   // GBK_TO_UNICODE[34568] := 16#E38B;
   // GBK_TO_UNICODE[34569] := 16#9292;
   // GBK_TO_UNICODE[34570] := 16#E38C;
   // GBK_TO_UNICODE[34571] := 16#9293;
   // GBK_TO_UNICODE[34572] := 16#E38D;
   // GBK_TO_UNICODE[34573] := 16#9294;
   // GBK_TO_UNICODE[34574] := 16#E38E;
   // GBK_TO_UNICODE[34575] := 16#9295;
   // GBK_TO_UNICODE[34576] := 16#E38F;
   // GBK_TO_UNICODE[34577] := 16#9296;
   // GBK_TO_UNICODE[34578] := 16#E390;
   // GBK_TO_UNICODE[34579] := 16#9297;
   // GBK_TO_UNICODE[34580] := 16#E391;
   // GBK_TO_UNICODE[34581] := 16#9298;
   // GBK_TO_UNICODE[34582] := 16#E392;
   // GBK_TO_UNICODE[34583] := 16#9299;
   // GBK_TO_UNICODE[34584] := 16#E393;
   // GBK_TO_UNICODE[34585] := 16#929A;
   // GBK_TO_UNICODE[34586] := 16#E394;
   // GBK_TO_UNICODE[34587] := 16#929B;
   // GBK_TO_UNICODE[34588] := 16#E395;
   // GBK_TO_UNICODE[34589] := 16#929C;
   // GBK_TO_UNICODE[34590] := 16#E396;
   // GBK_TO_UNICODE[34591] := 16#929D;
   // GBK_TO_UNICODE[34592] := 16#E397;
   // GBK_TO_UNICODE[34593] := 16#929E;
   // GBK_TO_UNICODE[34594] := 16#E398;
   // GBK_TO_UNICODE[34595] := 16#929F;
   // GBK_TO_UNICODE[34596] := 16#E399;
   // GBK_TO_UNICODE[34597] := 16#92A0;
   // GBK_TO_UNICODE[34598] := 16#E39A;
   // GBK_TO_UNICODE[34599] := 16#92A1;
   // GBK_TO_UNICODE[34600] := 16#E39B;
   // GBK_TO_UNICODE[34601] := 16#92A2;
   // GBK_TO_UNICODE[34602] := 16#E39C;
   // GBK_TO_UNICODE[34603] := 16#92A3;
   // GBK_TO_UNICODE[34604] := 16#E39D;
   // GBK_TO_UNICODE[34605] := 16#92A4;
   // GBK_TO_UNICODE[34606] := 16#E39E;
   // GBK_TO_UNICODE[34607] := 16#92A5;
   // GBK_TO_UNICODE[34608] := 16#E39F;
   // GBK_TO_UNICODE[34609] := 16#92A6;
   // GBK_TO_UNICODE[34610] := 16#E3A0;
   // GBK_TO_UNICODE[34611] := 16#92A7;
   // GBK_TO_UNICODE[34612] := 16#E3A1;
   // GBK_TO_UNICODE[34613] := 16#606A;
   // GBK_TO_UNICODE[34614] := 16#E3A2;
   // GBK_TO_UNICODE[34615] := 16#607D;
   // GBK_TO_UNICODE[34616] := 16#E3A3;
   // GBK_TO_UNICODE[34617] := 16#6096;
   // GBK_TO_UNICODE[34618] := 16#E3A4;
   // GBK_TO_UNICODE[34619] := 16#609A;
   // GBK_TO_UNICODE[34620] := 16#E3A5;
   // GBK_TO_UNICODE[34621] := 16#60AD;
   // GBK_TO_UNICODE[34622] := 16#E3A6;
   // GBK_TO_UNICODE[34623] := 16#609D;
   // GBK_TO_UNICODE[34624] := 16#E3A7;
   // GBK_TO_UNICODE[34625] := 16#6083;
   // GBK_TO_UNICODE[34626] := 16#E3A8;
   // GBK_TO_UNICODE[34627] := 16#6092;
   // GBK_TO_UNICODE[34628] := 16#E3A9;
   // GBK_TO_UNICODE[34629] := 16#608C;
   // GBK_TO_UNICODE[34630] := 16#E3AA;
   // GBK_TO_UNICODE[34631] := 16#609B;
   // GBK_TO_UNICODE[34632] := 16#E3AB;
   // GBK_TO_UNICODE[34633] := 16#60EC;
   // GBK_TO_UNICODE[34634] := 16#E3AC;
   // GBK_TO_UNICODE[34635] := 16#60BB;
   // GBK_TO_UNICODE[34636] := 16#E3AD;
   // GBK_TO_UNICODE[34637] := 16#60B1;
   // GBK_TO_UNICODE[34638] := 16#E3AE;
   // GBK_TO_UNICODE[34639] := 16#60DD;
   // GBK_TO_UNICODE[34640] := 16#E3AF;
   // GBK_TO_UNICODE[34641] := 16#60D8;
   // GBK_TO_UNICODE[34642] := 16#E3B0;
   // GBK_TO_UNICODE[34643] := 16#60C6;
   // GBK_TO_UNICODE[34644] := 16#E3B1;
   // GBK_TO_UNICODE[34645] := 16#60DA;
   // GBK_TO_UNICODE[34646] := 16#E3B2;
   // GBK_TO_UNICODE[34647] := 16#60B4;
   // GBK_TO_UNICODE[34648] := 16#E3B3;
   // GBK_TO_UNICODE[34649] := 16#6120;
   // GBK_TO_UNICODE[34650] := 16#E3B4;
   // GBK_TO_UNICODE[34651] := 16#6126;
   // GBK_TO_UNICODE[34652] := 16#E3B5;
   // GBK_TO_UNICODE[34653] := 16#6115;
   // GBK_TO_UNICODE[34654] := 16#E3B6;
   // GBK_TO_UNICODE[34655] := 16#6123;
   // GBK_TO_UNICODE[34656] := 16#E3B7;
   // GBK_TO_UNICODE[34657] := 16#60F4;
   // GBK_TO_UNICODE[34658] := 16#E3B8;
   // GBK_TO_UNICODE[34659] := 16#6100;
   // GBK_TO_UNICODE[34660] := 16#E3B9;
   // GBK_TO_UNICODE[34661] := 16#610E;
   // GBK_TO_UNICODE[34662] := 16#E3BA;
   // GBK_TO_UNICODE[34663] := 16#612B;
   // GBK_TO_UNICODE[34664] := 16#E3BB;
   // GBK_TO_UNICODE[34665] := 16#614A;
   // GBK_TO_UNICODE[34666] := 16#E3BC;
   // GBK_TO_UNICODE[34667] := 16#6175;
   // GBK_TO_UNICODE[34668] := 16#E3BD;
   // GBK_TO_UNICODE[34669] := 16#61AC;
   // GBK_TO_UNICODE[34670] := 16#E3BE;
   // GBK_TO_UNICODE[34671] := 16#6194;
   // GBK_TO_UNICODE[34672] := 16#E3BF;
   // GBK_TO_UNICODE[34673] := 16#61A7;
   // GBK_TO_UNICODE[34674] := 16#E3C0;
   // GBK_TO_UNICODE[34675] := 16#61B7;
   // GBK_TO_UNICODE[34676] := 16#E3C1;
   // GBK_TO_UNICODE[34677] := 16#61D4;
   // GBK_TO_UNICODE[34678] := 16#E3C2;
   // GBK_TO_UNICODE[34679] := 16#61F5;
   // GBK_TO_UNICODE[34680] := 16#E3C3;
   // GBK_TO_UNICODE[34681] := 16#5FDD;
   // GBK_TO_UNICODE[34682] := 16#E3C4;
   // GBK_TO_UNICODE[34683] := 16#96B3;
   // GBK_TO_UNICODE[34684] := 16#E3C5;
   // GBK_TO_UNICODE[34685] := 16#95E9;
   // GBK_TO_UNICODE[34686] := 16#E3C6;
   // GBK_TO_UNICODE[34687] := 16#95EB;
   // GBK_TO_UNICODE[34688] := 16#E3C7;
   // GBK_TO_UNICODE[34689] := 16#95F1;
   // GBK_TO_UNICODE[34690] := 16#E3C8;
   // GBK_TO_UNICODE[34691] := 16#95F3;
   // GBK_TO_UNICODE[34692] := 16#E3C9;
   // GBK_TO_UNICODE[34693] := 16#95F5;
   // GBK_TO_UNICODE[34694] := 16#E3CA;
   // GBK_TO_UNICODE[34695] := 16#95F6;
   // GBK_TO_UNICODE[34696] := 16#E3CB;
   // GBK_TO_UNICODE[34697] := 16#95FC;
   // GBK_TO_UNICODE[34698] := 16#E3CC;
   // GBK_TO_UNICODE[34699] := 16#95FE;
   // GBK_TO_UNICODE[34700] := 16#E3CD;
   // GBK_TO_UNICODE[34701] := 16#9603;
   // GBK_TO_UNICODE[34702] := 16#E3CE;
   // GBK_TO_UNICODE[34703] := 16#9604;
   // GBK_TO_UNICODE[34704] := 16#E3CF;
   // GBK_TO_UNICODE[34705] := 16#9606;
   // GBK_TO_UNICODE[34706] := 16#E3D0;
   // GBK_TO_UNICODE[34707] := 16#9608;
   // GBK_TO_UNICODE[34708] := 16#E3D1;
   // GBK_TO_UNICODE[34709] := 16#960A;
   // GBK_TO_UNICODE[34710] := 16#E3D2;
   // GBK_TO_UNICODE[34711] := 16#960B;
   // GBK_TO_UNICODE[34712] := 16#E3D3;
   // GBK_TO_UNICODE[34713] := 16#960C;
   // GBK_TO_UNICODE[34714] := 16#E3D4;
   // GBK_TO_UNICODE[34715] := 16#960D;
   // GBK_TO_UNICODE[34716] := 16#E3D5;
   // GBK_TO_UNICODE[34717] := 16#960F;
   // GBK_TO_UNICODE[34718] := 16#E3D6;
   // GBK_TO_UNICODE[34719] := 16#9612;
   // GBK_TO_UNICODE[34720] := 16#E3D7;
   // GBK_TO_UNICODE[34721] := 16#9615;
   // GBK_TO_UNICODE[34722] := 16#E3D8;
   // GBK_TO_UNICODE[34723] := 16#9616;
   // GBK_TO_UNICODE[34724] := 16#E3D9;
   // GBK_TO_UNICODE[34725] := 16#9617;
   // GBK_TO_UNICODE[34726] := 16#E3DA;
   // GBK_TO_UNICODE[34727] := 16#9619;
   // GBK_TO_UNICODE[34728] := 16#E3DB;
   // GBK_TO_UNICODE[34729] := 16#961A;
   // GBK_TO_UNICODE[34730] := 16#E3DC;
   // GBK_TO_UNICODE[34731] := 16#4E2C;
   // GBK_TO_UNICODE[34732] := 16#E3DD;
   // GBK_TO_UNICODE[34733] := 16#723F;
   // GBK_TO_UNICODE[34734] := 16#E3DE;
   // GBK_TO_UNICODE[34735] := 16#6215;
   // GBK_TO_UNICODE[34736] := 16#E3DF;
   // GBK_TO_UNICODE[34737] := 16#6C35;
   // GBK_TO_UNICODE[34738] := 16#E3E0;
   // GBK_TO_UNICODE[34739] := 16#6C54;
   // GBK_TO_UNICODE[34740] := 16#E3E1;
   // GBK_TO_UNICODE[34741] := 16#6C5C;
   // GBK_TO_UNICODE[34742] := 16#E3E2;
   // GBK_TO_UNICODE[34743] := 16#6C4A;
   // GBK_TO_UNICODE[34744] := 16#E3E3;
   // GBK_TO_UNICODE[34745] := 16#6CA3;
   // GBK_TO_UNICODE[34746] := 16#E3E4;
   // GBK_TO_UNICODE[34747] := 16#6C85;
   // GBK_TO_UNICODE[34748] := 16#E3E5;
   // GBK_TO_UNICODE[34749] := 16#6C90;
   // GBK_TO_UNICODE[34750] := 16#E3E6;
   // GBK_TO_UNICODE[34751] := 16#6C94;
   // GBK_TO_UNICODE[34752] := 16#E3E7;
   // GBK_TO_UNICODE[34753] := 16#6C8C;
   // GBK_TO_UNICODE[34754] := 16#E3E8;
   // GBK_TO_UNICODE[34755] := 16#6C68;
   // GBK_TO_UNICODE[34756] := 16#E3E9;
   // GBK_TO_UNICODE[34757] := 16#6C69;
   // GBK_TO_UNICODE[34758] := 16#E3EA;
   // GBK_TO_UNICODE[34759] := 16#6C74;
   // GBK_TO_UNICODE[34760] := 16#E3EB;
   // GBK_TO_UNICODE[34761] := 16#6C76;
   // GBK_TO_UNICODE[34762] := 16#E3EC;
   // GBK_TO_UNICODE[34763] := 16#6C86;
   // GBK_TO_UNICODE[34764] := 16#E3ED;
   // GBK_TO_UNICODE[34765] := 16#6CA9;
   // GBK_TO_UNICODE[34766] := 16#E3EE;
   // GBK_TO_UNICODE[34767] := 16#6CD0;
   // GBK_TO_UNICODE[34768] := 16#E3EF;
   // GBK_TO_UNICODE[34769] := 16#6CD4;
   // GBK_TO_UNICODE[34770] := 16#E3F0;
   // GBK_TO_UNICODE[34771] := 16#6CAD;
   // GBK_TO_UNICODE[34772] := 16#E3F1;
   // GBK_TO_UNICODE[34773] := 16#6CF7;
   // GBK_TO_UNICODE[34774] := 16#E3F2;
   // GBK_TO_UNICODE[34775] := 16#6CF8;
   // GBK_TO_UNICODE[34776] := 16#E3F3;
   // GBK_TO_UNICODE[34777] := 16#6CF1;
   // GBK_TO_UNICODE[34778] := 16#E3F4;
   // GBK_TO_UNICODE[34779] := 16#6CD7;
   // GBK_TO_UNICODE[34780] := 16#E3F5;
   // GBK_TO_UNICODE[34781] := 16#6CB2;
   // GBK_TO_UNICODE[34782] := 16#E3F6;
   // GBK_TO_UNICODE[34783] := 16#6CE0;
   // GBK_TO_UNICODE[34784] := 16#E3F7;
   // GBK_TO_UNICODE[34785] := 16#6CD6;
   // GBK_TO_UNICODE[34786] := 16#E3F8;
   // GBK_TO_UNICODE[34787] := 16#6CFA;
   // GBK_TO_UNICODE[34788] := 16#E3F9;
   // GBK_TO_UNICODE[34789] := 16#6CEB;
   // GBK_TO_UNICODE[34790] := 16#E3FA;
   // GBK_TO_UNICODE[34791] := 16#6CEE;
   // GBK_TO_UNICODE[34792] := 16#E3FB;
   // GBK_TO_UNICODE[34793] := 16#6CB1;
   // GBK_TO_UNICODE[34794] := 16#E3FC;
   // GBK_TO_UNICODE[34795] := 16#6CD3;
   // GBK_TO_UNICODE[34796] := 16#E3FD;
   // GBK_TO_UNICODE[34797] := 16#6CEF;
   // GBK_TO_UNICODE[34798] := 16#E3FE;
   // GBK_TO_UNICODE[34799] := 16#6CFE;
   // GBK_TO_UNICODE[34800] := 16#E440;
   // GBK_TO_UNICODE[34801] := 16#92A8;
   // GBK_TO_UNICODE[34802] := 16#E441;
   // GBK_TO_UNICODE[34803] := 16#92A9;
   // GBK_TO_UNICODE[34804] := 16#E442;
   // GBK_TO_UNICODE[34805] := 16#92AA;
   // GBK_TO_UNICODE[34806] := 16#E443;
   // GBK_TO_UNICODE[34807] := 16#92AB;
   // GBK_TO_UNICODE[34808] := 16#E444;
   // GBK_TO_UNICODE[34809] := 16#92AC;
   // GBK_TO_UNICODE[34810] := 16#E445;
   // GBK_TO_UNICODE[34811] := 16#92AD;
   // GBK_TO_UNICODE[34812] := 16#E446;
   // GBK_TO_UNICODE[34813] := 16#92AF;
   // GBK_TO_UNICODE[34814] := 16#E447;
   // GBK_TO_UNICODE[34815] := 16#92B0;
   // GBK_TO_UNICODE[34816] := 16#E448;
   // GBK_TO_UNICODE[34817] := 16#92B1;
   // GBK_TO_UNICODE[34818] := 16#E449;
   // GBK_TO_UNICODE[34819] := 16#92B2;
   // GBK_TO_UNICODE[34820] := 16#E44A;
   // GBK_TO_UNICODE[34821] := 16#92B3;
   // GBK_TO_UNICODE[34822] := 16#E44B;
   // GBK_TO_UNICODE[34823] := 16#92B4;
   // GBK_TO_UNICODE[34824] := 16#E44C;
   // GBK_TO_UNICODE[34825] := 16#92B5;
   // GBK_TO_UNICODE[34826] := 16#E44D;
   // GBK_TO_UNICODE[34827] := 16#92B6;
   // GBK_TO_UNICODE[34828] := 16#E44E;
   // GBK_TO_UNICODE[34829] := 16#92B7;
   // GBK_TO_UNICODE[34830] := 16#E44F;
   // GBK_TO_UNICODE[34831] := 16#92B8;
   // GBK_TO_UNICODE[34832] := 16#E450;
   // GBK_TO_UNICODE[34833] := 16#92B9;
   // GBK_TO_UNICODE[34834] := 16#E451;
   // GBK_TO_UNICODE[34835] := 16#92BA;
   // GBK_TO_UNICODE[34836] := 16#E452;
   // GBK_TO_UNICODE[34837] := 16#92BB;
   // GBK_TO_UNICODE[34838] := 16#E453;
   // GBK_TO_UNICODE[34839] := 16#92BC;
   // GBK_TO_UNICODE[34840] := 16#E454;
   // GBK_TO_UNICODE[34841] := 16#92BD;
   // GBK_TO_UNICODE[34842] := 16#E455;
   // GBK_TO_UNICODE[34843] := 16#92BE;
   // GBK_TO_UNICODE[34844] := 16#E456;
   // GBK_TO_UNICODE[34845] := 16#92BF;
   // GBK_TO_UNICODE[34846] := 16#E457;
   // GBK_TO_UNICODE[34847] := 16#92C0;
   // GBK_TO_UNICODE[34848] := 16#E458;
   // GBK_TO_UNICODE[34849] := 16#92C1;
   // GBK_TO_UNICODE[34850] := 16#E459;
   // GBK_TO_UNICODE[34851] := 16#92C2;
   // GBK_TO_UNICODE[34852] := 16#E45A;
   // GBK_TO_UNICODE[34853] := 16#92C3;
   // GBK_TO_UNICODE[34854] := 16#E45B;
   // GBK_TO_UNICODE[34855] := 16#92C4;
   // GBK_TO_UNICODE[34856] := 16#E45C;
   // GBK_TO_UNICODE[34857] := 16#92C5;
   // GBK_TO_UNICODE[34858] := 16#E45D;
   // GBK_TO_UNICODE[34859] := 16#92C6;
   // GBK_TO_UNICODE[34860] := 16#E45E;
   // GBK_TO_UNICODE[34861] := 16#92C7;
   // GBK_TO_UNICODE[34862] := 16#E45F;
   // GBK_TO_UNICODE[34863] := 16#92C9;
   // GBK_TO_UNICODE[34864] := 16#E460;
   // GBK_TO_UNICODE[34865] := 16#92CA;
   // GBK_TO_UNICODE[34866] := 16#E461;
   // GBK_TO_UNICODE[34867] := 16#92CB;
   // GBK_TO_UNICODE[34868] := 16#E462;
   // GBK_TO_UNICODE[34869] := 16#92CC;
   // GBK_TO_UNICODE[34870] := 16#E463;
   // GBK_TO_UNICODE[34871] := 16#92CD;
   // GBK_TO_UNICODE[34872] := 16#E464;
   // GBK_TO_UNICODE[34873] := 16#92CE;
   // GBK_TO_UNICODE[34874] := 16#E465;
   // GBK_TO_UNICODE[34875] := 16#92CF;
   // GBK_TO_UNICODE[34876] := 16#E466;
   // GBK_TO_UNICODE[34877] := 16#92D0;
   // GBK_TO_UNICODE[34878] := 16#E467;
   // GBK_TO_UNICODE[34879] := 16#92D1;
   // GBK_TO_UNICODE[34880] := 16#E468;
   // GBK_TO_UNICODE[34881] := 16#92D2;
   // GBK_TO_UNICODE[34882] := 16#E469;
   // GBK_TO_UNICODE[34883] := 16#92D3;
   // GBK_TO_UNICODE[34884] := 16#E46A;
   // GBK_TO_UNICODE[34885] := 16#92D4;
   // GBK_TO_UNICODE[34886] := 16#E46B;
   // GBK_TO_UNICODE[34887] := 16#92D5;
   // GBK_TO_UNICODE[34888] := 16#E46C;
   // GBK_TO_UNICODE[34889] := 16#92D6;
   // GBK_TO_UNICODE[34890] := 16#E46D;
   // GBK_TO_UNICODE[34891] := 16#92D7;
   // GBK_TO_UNICODE[34892] := 16#E46E;
   // GBK_TO_UNICODE[34893] := 16#92D8;
   // GBK_TO_UNICODE[34894] := 16#E46F;
   // GBK_TO_UNICODE[34895] := 16#92D9;
   // GBK_TO_UNICODE[34896] := 16#E470;
   // GBK_TO_UNICODE[34897] := 16#92DA;
   // GBK_TO_UNICODE[34898] := 16#E471;
   // GBK_TO_UNICODE[34899] := 16#92DB;
   // GBK_TO_UNICODE[34900] := 16#E472;
   // GBK_TO_UNICODE[34901] := 16#92DC;
   // GBK_TO_UNICODE[34902] := 16#E473;
   // GBK_TO_UNICODE[34903] := 16#92DD;
   // GBK_TO_UNICODE[34904] := 16#E474;
   // GBK_TO_UNICODE[34905] := 16#92DE;
   // GBK_TO_UNICODE[34906] := 16#E475;
   // GBK_TO_UNICODE[34907] := 16#92DF;
   // GBK_TO_UNICODE[34908] := 16#E476;
   // GBK_TO_UNICODE[34909] := 16#92E0;
   // GBK_TO_UNICODE[34910] := 16#E477;
   // GBK_TO_UNICODE[34911] := 16#92E1;
   // GBK_TO_UNICODE[34912] := 16#E478;
   // GBK_TO_UNICODE[34913] := 16#92E2;
   // GBK_TO_UNICODE[34914] := 16#E479;
   // GBK_TO_UNICODE[34915] := 16#92E3;
   // GBK_TO_UNICODE[34916] := 16#E47A;
   // GBK_TO_UNICODE[34917] := 16#92E4;
   // GBK_TO_UNICODE[34918] := 16#E47B;
   // GBK_TO_UNICODE[34919] := 16#92E5;
   // GBK_TO_UNICODE[34920] := 16#E47C;
   // GBK_TO_UNICODE[34921] := 16#92E6;
   // GBK_TO_UNICODE[34922] := 16#E47D;
   // GBK_TO_UNICODE[34923] := 16#92E7;
   // GBK_TO_UNICODE[34924] := 16#E47E;
   // GBK_TO_UNICODE[34925] := 16#92E8;
   // GBK_TO_UNICODE[34926] := 16#E480;
   // GBK_TO_UNICODE[34927] := 16#92E9;
   // GBK_TO_UNICODE[34928] := 16#E481;
   // GBK_TO_UNICODE[34929] := 16#92EA;
   // GBK_TO_UNICODE[34930] := 16#E482;
   // GBK_TO_UNICODE[34931] := 16#92EB;
   // GBK_TO_UNICODE[34932] := 16#E483;
   // GBK_TO_UNICODE[34933] := 16#92EC;
   // GBK_TO_UNICODE[34934] := 16#E484;
   // GBK_TO_UNICODE[34935] := 16#92ED;
   // GBK_TO_UNICODE[34936] := 16#E485;
   // GBK_TO_UNICODE[34937] := 16#92EE;
   // GBK_TO_UNICODE[34938] := 16#E486;
   // GBK_TO_UNICODE[34939] := 16#92EF;
   // GBK_TO_UNICODE[34940] := 16#E487;
   // GBK_TO_UNICODE[34941] := 16#92F0;
   // GBK_TO_UNICODE[34942] := 16#E488;
   // GBK_TO_UNICODE[34943] := 16#92F1;
   // GBK_TO_UNICODE[34944] := 16#E489;
   // GBK_TO_UNICODE[34945] := 16#92F2;
   // GBK_TO_UNICODE[34946] := 16#E48A;
   // GBK_TO_UNICODE[34947] := 16#92F3;
   // GBK_TO_UNICODE[34948] := 16#E48B;
   // GBK_TO_UNICODE[34949] := 16#92F4;
   // GBK_TO_UNICODE[34950] := 16#E48C;
   // GBK_TO_UNICODE[34951] := 16#92F5;
   // GBK_TO_UNICODE[34952] := 16#E48D;
   // GBK_TO_UNICODE[34953] := 16#92F6;
   // GBK_TO_UNICODE[34954] := 16#E48E;
   // GBK_TO_UNICODE[34955] := 16#92F7;
   // GBK_TO_UNICODE[34956] := 16#E48F;
   // GBK_TO_UNICODE[34957] := 16#92F8;
   // GBK_TO_UNICODE[34958] := 16#E490;
   // GBK_TO_UNICODE[34959] := 16#92F9;
   // GBK_TO_UNICODE[34960] := 16#E491;
   // GBK_TO_UNICODE[34961] := 16#92FA;
   // GBK_TO_UNICODE[34962] := 16#E492;
   // GBK_TO_UNICODE[34963] := 16#92FB;
   // GBK_TO_UNICODE[34964] := 16#E493;
   // GBK_TO_UNICODE[34965] := 16#92FC;
   // GBK_TO_UNICODE[34966] := 16#E494;
   // GBK_TO_UNICODE[34967] := 16#92FD;
   // GBK_TO_UNICODE[34968] := 16#E495;
   // GBK_TO_UNICODE[34969] := 16#92FE;
   // GBK_TO_UNICODE[34970] := 16#E496;
   // GBK_TO_UNICODE[34971] := 16#92FF;
   // GBK_TO_UNICODE[34972] := 16#E497;
   // GBK_TO_UNICODE[34973] := 16#9300;
   // GBK_TO_UNICODE[34974] := 16#E498;
   // GBK_TO_UNICODE[34975] := 16#9301;
   // GBK_TO_UNICODE[34976] := 16#E499;
   // GBK_TO_UNICODE[34977] := 16#9302;
   // GBK_TO_UNICODE[34978] := 16#E49A;
   // GBK_TO_UNICODE[34979] := 16#9303;
   // GBK_TO_UNICODE[34980] := 16#E49B;
   // GBK_TO_UNICODE[34981] := 16#9304;
   // GBK_TO_UNICODE[34982] := 16#E49C;
   // GBK_TO_UNICODE[34983] := 16#9305;
   // GBK_TO_UNICODE[34984] := 16#E49D;
   // GBK_TO_UNICODE[34985] := 16#9306;
   // GBK_TO_UNICODE[34986] := 16#E49E;
   // GBK_TO_UNICODE[34987] := 16#9307;
   // GBK_TO_UNICODE[34988] := 16#E49F;
   // GBK_TO_UNICODE[34989] := 16#9308;
   // GBK_TO_UNICODE[34990] := 16#E4A0;
   // GBK_TO_UNICODE[34991] := 16#9309;
   // GBK_TO_UNICODE[34992] := 16#E4A1;
   // GBK_TO_UNICODE[34993] := 16#6D39;
   // GBK_TO_UNICODE[34994] := 16#E4A2;
   // GBK_TO_UNICODE[34995] := 16#6D27;
   // GBK_TO_UNICODE[34996] := 16#E4A3;
   // GBK_TO_UNICODE[34997] := 16#6D0C;
   // GBK_TO_UNICODE[34998] := 16#E4A4;
   // GBK_TO_UNICODE[34999] := 16#6D43;
   // GBK_TO_UNICODE[35000] := 16#E4A5;
   // GBK_TO_UNICODE[35001] := 16#6D48;
   // GBK_TO_UNICODE[35002] := 16#E4A6;
   // GBK_TO_UNICODE[35003] := 16#6D07;
   // GBK_TO_UNICODE[35004] := 16#E4A7;
   // GBK_TO_UNICODE[35005] := 16#6D04;
   // GBK_TO_UNICODE[35006] := 16#E4A8;
   // GBK_TO_UNICODE[35007] := 16#6D19;
   // GBK_TO_UNICODE[35008] := 16#E4A9;
   // GBK_TO_UNICODE[35009] := 16#6D0E;
   // GBK_TO_UNICODE[35010] := 16#E4AA;
   // GBK_TO_UNICODE[35011] := 16#6D2B;
   // GBK_TO_UNICODE[35012] := 16#E4AB;
   // GBK_TO_UNICODE[35013] := 16#6D4D;
   // GBK_TO_UNICODE[35014] := 16#E4AC;
   // GBK_TO_UNICODE[35015] := 16#6D2E;
   // GBK_TO_UNICODE[35016] := 16#E4AD;
   // GBK_TO_UNICODE[35017] := 16#6D35;
   // GBK_TO_UNICODE[35018] := 16#E4AE;
   // GBK_TO_UNICODE[35019] := 16#6D1A;
   // GBK_TO_UNICODE[35020] := 16#E4AF;
   // GBK_TO_UNICODE[35021] := 16#6D4F;
   // GBK_TO_UNICODE[35022] := 16#E4B0;
   // GBK_TO_UNICODE[35023] := 16#6D52;
   // GBK_TO_UNICODE[35024] := 16#E4B1;
   // GBK_TO_UNICODE[35025] := 16#6D54;
   // GBK_TO_UNICODE[35026] := 16#E4B2;
   // GBK_TO_UNICODE[35027] := 16#6D33;
   // GBK_TO_UNICODE[35028] := 16#E4B3;
   // GBK_TO_UNICODE[35029] := 16#6D91;
   // GBK_TO_UNICODE[35030] := 16#E4B4;
   // GBK_TO_UNICODE[35031] := 16#6D6F;
   // GBK_TO_UNICODE[35032] := 16#E4B5;
   // GBK_TO_UNICODE[35033] := 16#6D9E;
   // GBK_TO_UNICODE[35034] := 16#E4B6;
   // GBK_TO_UNICODE[35035] := 16#6DA0;
   // GBK_TO_UNICODE[35036] := 16#E4B7;
   // GBK_TO_UNICODE[35037] := 16#6D5E;
   // GBK_TO_UNICODE[35038] := 16#E4B8;
   // GBK_TO_UNICODE[35039] := 16#6D93;
   // GBK_TO_UNICODE[35040] := 16#E4B9;
   // GBK_TO_UNICODE[35041] := 16#6D94;
   // GBK_TO_UNICODE[35042] := 16#E4BA;
   // GBK_TO_UNICODE[35043] := 16#6D5C;
   // GBK_TO_UNICODE[35044] := 16#E4BB;
   // GBK_TO_UNICODE[35045] := 16#6D60;
   // GBK_TO_UNICODE[35046] := 16#E4BC;
   // GBK_TO_UNICODE[35047] := 16#6D7C;
   // GBK_TO_UNICODE[35048] := 16#E4BD;
   // GBK_TO_UNICODE[35049] := 16#6D63;
   // GBK_TO_UNICODE[35050] := 16#E4BE;
   // GBK_TO_UNICODE[35051] := 16#6E1A;
   // GBK_TO_UNICODE[35052] := 16#E4BF;
   // GBK_TO_UNICODE[35053] := 16#6DC7;
   // GBK_TO_UNICODE[35054] := 16#E4C0;
   // GBK_TO_UNICODE[35055] := 16#6DC5;
   // GBK_TO_UNICODE[35056] := 16#E4C1;
   // GBK_TO_UNICODE[35057] := 16#6DDE;
   // GBK_TO_UNICODE[35058] := 16#E4C2;
   // GBK_TO_UNICODE[35059] := 16#6E0E;
   // GBK_TO_UNICODE[35060] := 16#E4C3;
   // GBK_TO_UNICODE[35061] := 16#6DBF;
   // GBK_TO_UNICODE[35062] := 16#E4C4;
   // GBK_TO_UNICODE[35063] := 16#6DE0;
   // GBK_TO_UNICODE[35064] := 16#E4C5;
   // GBK_TO_UNICODE[35065] := 16#6E11;
   // GBK_TO_UNICODE[35066] := 16#E4C6;
   // GBK_TO_UNICODE[35067] := 16#6DE6;
   // GBK_TO_UNICODE[35068] := 16#E4C7;
   // GBK_TO_UNICODE[35069] := 16#6DDD;
   // GBK_TO_UNICODE[35070] := 16#E4C8;
   // GBK_TO_UNICODE[35071] := 16#6DD9;
   // GBK_TO_UNICODE[35072] := 16#E4C9;
   // GBK_TO_UNICODE[35073] := 16#6E16;
   // GBK_TO_UNICODE[35074] := 16#E4CA;
   // GBK_TO_UNICODE[35075] := 16#6DAB;
   // GBK_TO_UNICODE[35076] := 16#E4CB;
   // GBK_TO_UNICODE[35077] := 16#6E0C;
   // GBK_TO_UNICODE[35078] := 16#E4CC;
   // GBK_TO_UNICODE[35079] := 16#6DAE;
   // GBK_TO_UNICODE[35080] := 16#E4CD;
   // GBK_TO_UNICODE[35081] := 16#6E2B;
   // GBK_TO_UNICODE[35082] := 16#E4CE;
   // GBK_TO_UNICODE[35083] := 16#6E6E;
   // GBK_TO_UNICODE[35084] := 16#E4CF;
   // GBK_TO_UNICODE[35085] := 16#6E4E;
   // GBK_TO_UNICODE[35086] := 16#E4D0;
   // GBK_TO_UNICODE[35087] := 16#6E6B;
   // GBK_TO_UNICODE[35088] := 16#E4D1;
   // GBK_TO_UNICODE[35089] := 16#6EB2;
   // GBK_TO_UNICODE[35090] := 16#E4D2;
   // GBK_TO_UNICODE[35091] := 16#6E5F;
   // GBK_TO_UNICODE[35092] := 16#E4D3;
   // GBK_TO_UNICODE[35093] := 16#6E86;
   // GBK_TO_UNICODE[35094] := 16#E4D4;
   // GBK_TO_UNICODE[35095] := 16#6E53;
   // GBK_TO_UNICODE[35096] := 16#E4D5;
   // GBK_TO_UNICODE[35097] := 16#6E54;
   // GBK_TO_UNICODE[35098] := 16#E4D6;
   // GBK_TO_UNICODE[35099] := 16#6E32;
   // GBK_TO_UNICODE[35100] := 16#E4D7;
   // GBK_TO_UNICODE[35101] := 16#6E25;
   // GBK_TO_UNICODE[35102] := 16#E4D8;
   // GBK_TO_UNICODE[35103] := 16#6E44;
   // GBK_TO_UNICODE[35104] := 16#E4D9;
   // GBK_TO_UNICODE[35105] := 16#6EDF;
   // GBK_TO_UNICODE[35106] := 16#E4DA;
   // GBK_TO_UNICODE[35107] := 16#6EB1;
   // GBK_TO_UNICODE[35108] := 16#E4DB;
   // GBK_TO_UNICODE[35109] := 16#6E98;
   // GBK_TO_UNICODE[35110] := 16#E4DC;
   // GBK_TO_UNICODE[35111] := 16#6EE0;
   // GBK_TO_UNICODE[35112] := 16#E4DD;
   // GBK_TO_UNICODE[35113] := 16#6F2D;
   // GBK_TO_UNICODE[35114] := 16#E4DE;
   // GBK_TO_UNICODE[35115] := 16#6EE2;
   // GBK_TO_UNICODE[35116] := 16#E4DF;
   // GBK_TO_UNICODE[35117] := 16#6EA5;
   // GBK_TO_UNICODE[35118] := 16#E4E0;
   // GBK_TO_UNICODE[35119] := 16#6EA7;
   // GBK_TO_UNICODE[35120] := 16#E4E1;
   // GBK_TO_UNICODE[35121] := 16#6EBD;
   // GBK_TO_UNICODE[35122] := 16#E4E2;
   // GBK_TO_UNICODE[35123] := 16#6EBB;
   // GBK_TO_UNICODE[35124] := 16#E4E3;
   // GBK_TO_UNICODE[35125] := 16#6EB7;
   // GBK_TO_UNICODE[35126] := 16#E4E4;
   // GBK_TO_UNICODE[35127] := 16#6ED7;
   // GBK_TO_UNICODE[35128] := 16#E4E5;
   // GBK_TO_UNICODE[35129] := 16#6EB4;
   // GBK_TO_UNICODE[35130] := 16#E4E6;
   // GBK_TO_UNICODE[35131] := 16#6ECF;
   // GBK_TO_UNICODE[35132] := 16#E4E7;
   // GBK_TO_UNICODE[35133] := 16#6E8F;
   // GBK_TO_UNICODE[35134] := 16#E4E8;
   // GBK_TO_UNICODE[35135] := 16#6EC2;
   // GBK_TO_UNICODE[35136] := 16#E4E9;
   // GBK_TO_UNICODE[35137] := 16#6E9F;
   // GBK_TO_UNICODE[35138] := 16#E4EA;
   // GBK_TO_UNICODE[35139] := 16#6F62;
   // GBK_TO_UNICODE[35140] := 16#E4EB;
   // GBK_TO_UNICODE[35141] := 16#6F46;
   // GBK_TO_UNICODE[35142] := 16#E4EC;
   // GBK_TO_UNICODE[35143] := 16#6F47;
   // GBK_TO_UNICODE[35144] := 16#E4ED;
   // GBK_TO_UNICODE[35145] := 16#6F24;
   // GBK_TO_UNICODE[35146] := 16#E4EE;
   // GBK_TO_UNICODE[35147] := 16#6F15;
   // GBK_TO_UNICODE[35148] := 16#E4EF;
   // GBK_TO_UNICODE[35149] := 16#6EF9;
   // GBK_TO_UNICODE[35150] := 16#E4F0;
   // GBK_TO_UNICODE[35151] := 16#6F2F;
   // GBK_TO_UNICODE[35152] := 16#E4F1;
   // GBK_TO_UNICODE[35153] := 16#6F36;
   // GBK_TO_UNICODE[35154] := 16#E4F2;
   // GBK_TO_UNICODE[35155] := 16#6F4B;
   // GBK_TO_UNICODE[35156] := 16#E4F3;
   // GBK_TO_UNICODE[35157] := 16#6F74;
   // GBK_TO_UNICODE[35158] := 16#E4F4;
   // GBK_TO_UNICODE[35159] := 16#6F2A;
   // GBK_TO_UNICODE[35160] := 16#E4F5;
   // GBK_TO_UNICODE[35161] := 16#6F09;
   // GBK_TO_UNICODE[35162] := 16#E4F6;
   // GBK_TO_UNICODE[35163] := 16#6F29;
   // GBK_TO_UNICODE[35164] := 16#E4F7;
   // GBK_TO_UNICODE[35165] := 16#6F89;
   // GBK_TO_UNICODE[35166] := 16#E4F8;
   // GBK_TO_UNICODE[35167] := 16#6F8D;
   // GBK_TO_UNICODE[35168] := 16#E4F9;
   // GBK_TO_UNICODE[35169] := 16#6F8C;
   // GBK_TO_UNICODE[35170] := 16#E4FA;
   // GBK_TO_UNICODE[35171] := 16#6F78;
   // GBK_TO_UNICODE[35172] := 16#E4FB;
   // GBK_TO_UNICODE[35173] := 16#6F72;
   // GBK_TO_UNICODE[35174] := 16#E4FC;
   // GBK_TO_UNICODE[35175] := 16#6F7C;
   // GBK_TO_UNICODE[35176] := 16#E4FD;
   // GBK_TO_UNICODE[35177] := 16#6F7A;
   // GBK_TO_UNICODE[35178] := 16#E4FE;
   // GBK_TO_UNICODE[35179] := 16#6FD1;
   // GBK_TO_UNICODE[35180] := 16#E540;
   // GBK_TO_UNICODE[35181] := 16#930A;
   // GBK_TO_UNICODE[35182] := 16#E541;
   // GBK_TO_UNICODE[35183] := 16#930B;
   // GBK_TO_UNICODE[35184] := 16#E542;
   // GBK_TO_UNICODE[35185] := 16#930C;
   // GBK_TO_UNICODE[35186] := 16#E543;
   // GBK_TO_UNICODE[35187] := 16#930D;
   // GBK_TO_UNICODE[35188] := 16#E544;
   // GBK_TO_UNICODE[35189] := 16#930E;
   // GBK_TO_UNICODE[35190] := 16#E545;
   // GBK_TO_UNICODE[35191] := 16#930F;
   // GBK_TO_UNICODE[35192] := 16#E546;
   // GBK_TO_UNICODE[35193] := 16#9310;
   // GBK_TO_UNICODE[35194] := 16#E547;
   // GBK_TO_UNICODE[35195] := 16#9311;
   // GBK_TO_UNICODE[35196] := 16#E548;
   // GBK_TO_UNICODE[35197] := 16#9312;
   // GBK_TO_UNICODE[35198] := 16#E549;
   // GBK_TO_UNICODE[35199] := 16#9313;
   // GBK_TO_UNICODE[35200] := 16#E54A;
   // GBK_TO_UNICODE[35201] := 16#9314;
   // GBK_TO_UNICODE[35202] := 16#E54B;
   // GBK_TO_UNICODE[35203] := 16#9315;
   // GBK_TO_UNICODE[35204] := 16#E54C;
   // GBK_TO_UNICODE[35205] := 16#9316;
   // GBK_TO_UNICODE[35206] := 16#E54D;
   // GBK_TO_UNICODE[35207] := 16#9317;
   // GBK_TO_UNICODE[35208] := 16#E54E;
   // GBK_TO_UNICODE[35209] := 16#9318;
   // GBK_TO_UNICODE[35210] := 16#E54F;
   // GBK_TO_UNICODE[35211] := 16#9319;
   // GBK_TO_UNICODE[35212] := 16#E550;
   // GBK_TO_UNICODE[35213] := 16#931A;
   // GBK_TO_UNICODE[35214] := 16#E551;
   // GBK_TO_UNICODE[35215] := 16#931B;
   // GBK_TO_UNICODE[35216] := 16#E552;
   // GBK_TO_UNICODE[35217] := 16#931C;
   // GBK_TO_UNICODE[35218] := 16#E553;
   // GBK_TO_UNICODE[35219] := 16#931D;
   // GBK_TO_UNICODE[35220] := 16#E554;
   // GBK_TO_UNICODE[35221] := 16#931E;
   // GBK_TO_UNICODE[35222] := 16#E555;
   // GBK_TO_UNICODE[35223] := 16#931F;
   // GBK_TO_UNICODE[35224] := 16#E556;
   // GBK_TO_UNICODE[35225] := 16#9320;
   // GBK_TO_UNICODE[35226] := 16#E557;
   // GBK_TO_UNICODE[35227] := 16#9321;
   // GBK_TO_UNICODE[35228] := 16#E558;
   // GBK_TO_UNICODE[35229] := 16#9322;
   // GBK_TO_UNICODE[35230] := 16#E559;
   // GBK_TO_UNICODE[35231] := 16#9323;
   // GBK_TO_UNICODE[35232] := 16#E55A;
   // GBK_TO_UNICODE[35233] := 16#9324;
   // GBK_TO_UNICODE[35234] := 16#E55B;
   // GBK_TO_UNICODE[35235] := 16#9325;
   // GBK_TO_UNICODE[35236] := 16#E55C;
   // GBK_TO_UNICODE[35237] := 16#9326;
   // GBK_TO_UNICODE[35238] := 16#E55D;
   // GBK_TO_UNICODE[35239] := 16#9327;
   // GBK_TO_UNICODE[35240] := 16#E55E;
   // GBK_TO_UNICODE[35241] := 16#9328;
   // GBK_TO_UNICODE[35242] := 16#E55F;
   // GBK_TO_UNICODE[35243] := 16#9329;
   // GBK_TO_UNICODE[35244] := 16#E560;
   // GBK_TO_UNICODE[35245] := 16#932A;
   // GBK_TO_UNICODE[35246] := 16#E561;
   // GBK_TO_UNICODE[35247] := 16#932B;
   // GBK_TO_UNICODE[35248] := 16#E562;
   // GBK_TO_UNICODE[35249] := 16#932C;
   // GBK_TO_UNICODE[35250] := 16#E563;
   // GBK_TO_UNICODE[35251] := 16#932D;
   // GBK_TO_UNICODE[35252] := 16#E564;
   // GBK_TO_UNICODE[35253] := 16#932E;
   // GBK_TO_UNICODE[35254] := 16#E565;
   // GBK_TO_UNICODE[35255] := 16#932F;
   // GBK_TO_UNICODE[35256] := 16#E566;
   // GBK_TO_UNICODE[35257] := 16#9330;
   // GBK_TO_UNICODE[35258] := 16#E567;
   // GBK_TO_UNICODE[35259] := 16#9331;
   // GBK_TO_UNICODE[35260] := 16#E568;
   // GBK_TO_UNICODE[35261] := 16#9332;
   // GBK_TO_UNICODE[35262] := 16#E569;
   // GBK_TO_UNICODE[35263] := 16#9333;
   // GBK_TO_UNICODE[35264] := 16#E56A;
   // GBK_TO_UNICODE[35265] := 16#9334;
   // GBK_TO_UNICODE[35266] := 16#E56B;
   // GBK_TO_UNICODE[35267] := 16#9335;
   // GBK_TO_UNICODE[35268] := 16#E56C;
   // GBK_TO_UNICODE[35269] := 16#9336;
   // GBK_TO_UNICODE[35270] := 16#E56D;
   // GBK_TO_UNICODE[35271] := 16#9337;
   // GBK_TO_UNICODE[35272] := 16#E56E;
   // GBK_TO_UNICODE[35273] := 16#9338;
   // GBK_TO_UNICODE[35274] := 16#E56F;
   // GBK_TO_UNICODE[35275] := 16#9339;
   // GBK_TO_UNICODE[35276] := 16#E570;
   // GBK_TO_UNICODE[35277] := 16#933A;
   // GBK_TO_UNICODE[35278] := 16#E571;
   // GBK_TO_UNICODE[35279] := 16#933B;
   // GBK_TO_UNICODE[35280] := 16#E572;
   // GBK_TO_UNICODE[35281] := 16#933C;
   // GBK_TO_UNICODE[35282] := 16#E573;
   // GBK_TO_UNICODE[35283] := 16#933D;
   // GBK_TO_UNICODE[35284] := 16#E574;
   // GBK_TO_UNICODE[35285] := 16#933F;
   // GBK_TO_UNICODE[35286] := 16#E575;
   // GBK_TO_UNICODE[35287] := 16#9340;
   // GBK_TO_UNICODE[35288] := 16#E576;
   // GBK_TO_UNICODE[35289] := 16#9341;
   // GBK_TO_UNICODE[35290] := 16#E577;
   // GBK_TO_UNICODE[35291] := 16#9342;
   // GBK_TO_UNICODE[35292] := 16#E578;
   // GBK_TO_UNICODE[35293] := 16#9343;
   // GBK_TO_UNICODE[35294] := 16#E579;
   // GBK_TO_UNICODE[35295] := 16#9344;
   // GBK_TO_UNICODE[35296] := 16#E57A;
   // GBK_TO_UNICODE[35297] := 16#9345;
   // GBK_TO_UNICODE[35298] := 16#E57B;
   // GBK_TO_UNICODE[35299] := 16#9346;
   // GBK_TO_UNICODE[35300] := 16#E57C;
   // GBK_TO_UNICODE[35301] := 16#9347;
   // GBK_TO_UNICODE[35302] := 16#E57D;
   // GBK_TO_UNICODE[35303] := 16#9348;
   // GBK_TO_UNICODE[35304] := 16#E57E;
   // GBK_TO_UNICODE[35305] := 16#9349;
   // GBK_TO_UNICODE[35306] := 16#E580;
   // GBK_TO_UNICODE[35307] := 16#934A;
   // GBK_TO_UNICODE[35308] := 16#E581;
   // GBK_TO_UNICODE[35309] := 16#934B;
   // GBK_TO_UNICODE[35310] := 16#E582;
   // GBK_TO_UNICODE[35311] := 16#934C;
   // GBK_TO_UNICODE[35312] := 16#E583;
   // GBK_TO_UNICODE[35313] := 16#934D;
   // GBK_TO_UNICODE[35314] := 16#E584;
   // GBK_TO_UNICODE[35315] := 16#934E;
   // GBK_TO_UNICODE[35316] := 16#E585;
   // GBK_TO_UNICODE[35317] := 16#934F;
   // GBK_TO_UNICODE[35318] := 16#E586;
   // GBK_TO_UNICODE[35319] := 16#9350;
   // GBK_TO_UNICODE[35320] := 16#E587;
   // GBK_TO_UNICODE[35321] := 16#9351;
   // GBK_TO_UNICODE[35322] := 16#E588;
   // GBK_TO_UNICODE[35323] := 16#9352;
   // GBK_TO_UNICODE[35324] := 16#E589;
   // GBK_TO_UNICODE[35325] := 16#9353;
   // GBK_TO_UNICODE[35326] := 16#E58A;
   // GBK_TO_UNICODE[35327] := 16#9354;
   // GBK_TO_UNICODE[35328] := 16#E58B;
   // GBK_TO_UNICODE[35329] := 16#9355;
   // GBK_TO_UNICODE[35330] := 16#E58C;
   // GBK_TO_UNICODE[35331] := 16#9356;
   // GBK_TO_UNICODE[35332] := 16#E58D;
   // GBK_TO_UNICODE[35333] := 16#9357;
   // GBK_TO_UNICODE[35334] := 16#E58E;
   // GBK_TO_UNICODE[35335] := 16#9358;
   // GBK_TO_UNICODE[35336] := 16#E58F;
   // GBK_TO_UNICODE[35337] := 16#9359;
   // GBK_TO_UNICODE[35338] := 16#E590;
   // GBK_TO_UNICODE[35339] := 16#935A;
   // GBK_TO_UNICODE[35340] := 16#E591;
   // GBK_TO_UNICODE[35341] := 16#935B;
   // GBK_TO_UNICODE[35342] := 16#E592;
   // GBK_TO_UNICODE[35343] := 16#935C;
   // GBK_TO_UNICODE[35344] := 16#E593;
   // GBK_TO_UNICODE[35345] := 16#935D;
   // GBK_TO_UNICODE[35346] := 16#E594;
   // GBK_TO_UNICODE[35347] := 16#935E;
   // GBK_TO_UNICODE[35348] := 16#E595;
   // GBK_TO_UNICODE[35349] := 16#935F;
   // GBK_TO_UNICODE[35350] := 16#E596;
   // GBK_TO_UNICODE[35351] := 16#9360;
   // GBK_TO_UNICODE[35352] := 16#E597;
   // GBK_TO_UNICODE[35353] := 16#9361;
   // GBK_TO_UNICODE[35354] := 16#E598;
   // GBK_TO_UNICODE[35355] := 16#9362;
   // GBK_TO_UNICODE[35356] := 16#E599;
   // GBK_TO_UNICODE[35357] := 16#9363;
   // GBK_TO_UNICODE[35358] := 16#E59A;
   // GBK_TO_UNICODE[35359] := 16#9364;
   // GBK_TO_UNICODE[35360] := 16#E59B;
   // GBK_TO_UNICODE[35361] := 16#9365;
   // GBK_TO_UNICODE[35362] := 16#E59C;
   // GBK_TO_UNICODE[35363] := 16#9366;
   // GBK_TO_UNICODE[35364] := 16#E59D;
   // GBK_TO_UNICODE[35365] := 16#9367;
   // GBK_TO_UNICODE[35366] := 16#E59E;
   // GBK_TO_UNICODE[35367] := 16#9368;
   // GBK_TO_UNICODE[35368] := 16#E59F;
   // GBK_TO_UNICODE[35369] := 16#9369;
   // GBK_TO_UNICODE[35370] := 16#E5A0;
   // GBK_TO_UNICODE[35371] := 16#936B;
   // GBK_TO_UNICODE[35372] := 16#E5A1;
   // GBK_TO_UNICODE[35373] := 16#6FC9;
   // GBK_TO_UNICODE[35374] := 16#E5A2;
   // GBK_TO_UNICODE[35375] := 16#6FA7;
   // GBK_TO_UNICODE[35376] := 16#E5A3;
   // GBK_TO_UNICODE[35377] := 16#6FB9;
   // GBK_TO_UNICODE[35378] := 16#E5A4;
   // GBK_TO_UNICODE[35379] := 16#6FB6;
   // GBK_TO_UNICODE[35380] := 16#E5A5;
   // GBK_TO_UNICODE[35381] := 16#6FC2;
   // GBK_TO_UNICODE[35382] := 16#E5A6;
   // GBK_TO_UNICODE[35383] := 16#6FE1;
   // GBK_TO_UNICODE[35384] := 16#E5A7;
   // GBK_TO_UNICODE[35385] := 16#6FEE;
   // GBK_TO_UNICODE[35386] := 16#E5A8;
   // GBK_TO_UNICODE[35387] := 16#6FDE;
   // GBK_TO_UNICODE[35388] := 16#E5A9;
   // GBK_TO_UNICODE[35389] := 16#6FE0;
   // GBK_TO_UNICODE[35390] := 16#E5AA;
   // GBK_TO_UNICODE[35391] := 16#6FEF;
   // GBK_TO_UNICODE[35392] := 16#E5AB;
   // GBK_TO_UNICODE[35393] := 16#701A;
   // GBK_TO_UNICODE[35394] := 16#E5AC;
   // GBK_TO_UNICODE[35395] := 16#7023;
   // GBK_TO_UNICODE[35396] := 16#E5AD;
   // GBK_TO_UNICODE[35397] := 16#701B;
   // GBK_TO_UNICODE[35398] := 16#E5AE;
   // GBK_TO_UNICODE[35399] := 16#7039;
   // GBK_TO_UNICODE[35400] := 16#E5AF;
   // GBK_TO_UNICODE[35401] := 16#7035;
   // GBK_TO_UNICODE[35402] := 16#E5B0;
   // GBK_TO_UNICODE[35403] := 16#704F;
   // GBK_TO_UNICODE[35404] := 16#E5B1;
   // GBK_TO_UNICODE[35405] := 16#705E;
   // GBK_TO_UNICODE[35406] := 16#E5B2;
   // GBK_TO_UNICODE[35407] := 16#5B80;
   // GBK_TO_UNICODE[35408] := 16#E5B3;
   // GBK_TO_UNICODE[35409] := 16#5B84;
   // GBK_TO_UNICODE[35410] := 16#E5B4;
   // GBK_TO_UNICODE[35411] := 16#5B95;
   // GBK_TO_UNICODE[35412] := 16#E5B5;
   // GBK_TO_UNICODE[35413] := 16#5B93;
   // GBK_TO_UNICODE[35414] := 16#E5B6;
   // GBK_TO_UNICODE[35415] := 16#5BA5;
   // GBK_TO_UNICODE[35416] := 16#E5B7;
   // GBK_TO_UNICODE[35417] := 16#5BB8;
   // GBK_TO_UNICODE[35418] := 16#E5B8;
   // GBK_TO_UNICODE[35419] := 16#752F;
   // GBK_TO_UNICODE[35420] := 16#E5B9;
   // GBK_TO_UNICODE[35421] := 16#9A9E;
   // GBK_TO_UNICODE[35422] := 16#E5BA;
   // GBK_TO_UNICODE[35423] := 16#6434;
   // GBK_TO_UNICODE[35424] := 16#E5BB;
   // GBK_TO_UNICODE[35425] := 16#5BE4;
   // GBK_TO_UNICODE[35426] := 16#E5BC;
   // GBK_TO_UNICODE[35427] := 16#5BEE;
   // GBK_TO_UNICODE[35428] := 16#E5BD;
   // GBK_TO_UNICODE[35429] := 16#8930;
   // GBK_TO_UNICODE[35430] := 16#E5BE;
   // GBK_TO_UNICODE[35431] := 16#5BF0;
   // GBK_TO_UNICODE[35432] := 16#E5BF;
   // GBK_TO_UNICODE[35433] := 16#8E47;
   // GBK_TO_UNICODE[35434] := 16#E5C0;
   // GBK_TO_UNICODE[35435] := 16#8B07;
   // GBK_TO_UNICODE[35436] := 16#E5C1;
   // GBK_TO_UNICODE[35437] := 16#8FB6;
   // GBK_TO_UNICODE[35438] := 16#E5C2;
   // GBK_TO_UNICODE[35439] := 16#8FD3;
   // GBK_TO_UNICODE[35440] := 16#E5C3;
   // GBK_TO_UNICODE[35441] := 16#8FD5;
   // GBK_TO_UNICODE[35442] := 16#E5C4;
   // GBK_TO_UNICODE[35443] := 16#8FE5;
   // GBK_TO_UNICODE[35444] := 16#E5C5;
   // GBK_TO_UNICODE[35445] := 16#8FEE;
   // GBK_TO_UNICODE[35446] := 16#E5C6;
   // GBK_TO_UNICODE[35447] := 16#8FE4;
   // GBK_TO_UNICODE[35448] := 16#E5C7;
   // GBK_TO_UNICODE[35449] := 16#8FE9;
   // GBK_TO_UNICODE[35450] := 16#E5C8;
   // GBK_TO_UNICODE[35451] := 16#8FE6;
   // GBK_TO_UNICODE[35452] := 16#E5C9;
   // GBK_TO_UNICODE[35453] := 16#8FF3;
   // GBK_TO_UNICODE[35454] := 16#E5CA;
   // GBK_TO_UNICODE[35455] := 16#8FE8;
   // GBK_TO_UNICODE[35456] := 16#E5CB;
   // GBK_TO_UNICODE[35457] := 16#9005;
   // GBK_TO_UNICODE[35458] := 16#E5CC;
   // GBK_TO_UNICODE[35459] := 16#9004;
   // GBK_TO_UNICODE[35460] := 16#E5CD;
   // GBK_TO_UNICODE[35461] := 16#900B;
   // GBK_TO_UNICODE[35462] := 16#E5CE;
   // GBK_TO_UNICODE[35463] := 16#9026;
   // GBK_TO_UNICODE[35464] := 16#E5CF;
   // GBK_TO_UNICODE[35465] := 16#9011;
   // GBK_TO_UNICODE[35466] := 16#E5D0;
   // GBK_TO_UNICODE[35467] := 16#900D;
   // GBK_TO_UNICODE[35468] := 16#E5D1;
   // GBK_TO_UNICODE[35469] := 16#9016;
   // GBK_TO_UNICODE[35470] := 16#E5D2;
   // GBK_TO_UNICODE[35471] := 16#9021;
   // GBK_TO_UNICODE[35472] := 16#E5D3;
   // GBK_TO_UNICODE[35473] := 16#9035;
   // GBK_TO_UNICODE[35474] := 16#E5D4;
   // GBK_TO_UNICODE[35475] := 16#9036;
   // GBK_TO_UNICODE[35476] := 16#E5D5;
   // GBK_TO_UNICODE[35477] := 16#902D;
   // GBK_TO_UNICODE[35478] := 16#E5D6;
   // GBK_TO_UNICODE[35479] := 16#902F;
   // GBK_TO_UNICODE[35480] := 16#E5D7;
   // GBK_TO_UNICODE[35481] := 16#9044;
   // GBK_TO_UNICODE[35482] := 16#E5D8;
   // GBK_TO_UNICODE[35483] := 16#9051;
   // GBK_TO_UNICODE[35484] := 16#E5D9;
   // GBK_TO_UNICODE[35485] := 16#9052;
   // GBK_TO_UNICODE[35486] := 16#E5DA;
   // GBK_TO_UNICODE[35487] := 16#9050;
   // GBK_TO_UNICODE[35488] := 16#E5DB;
   // GBK_TO_UNICODE[35489] := 16#9068;
   // GBK_TO_UNICODE[35490] := 16#E5DC;
   // GBK_TO_UNICODE[35491] := 16#9058;
   // GBK_TO_UNICODE[35492] := 16#E5DD;
   // GBK_TO_UNICODE[35493] := 16#9062;
   // GBK_TO_UNICODE[35494] := 16#E5DE;
   // GBK_TO_UNICODE[35495] := 16#905B;
   // GBK_TO_UNICODE[35496] := 16#E5DF;
   // GBK_TO_UNICODE[35497] := 16#66B9;
   // GBK_TO_UNICODE[35498] := 16#E5E0;
   // GBK_TO_UNICODE[35499] := 16#9074;
   // GBK_TO_UNICODE[35500] := 16#E5E1;
   // GBK_TO_UNICODE[35501] := 16#907D;
   // GBK_TO_UNICODE[35502] := 16#E5E2;
   // GBK_TO_UNICODE[35503] := 16#9082;
   // GBK_TO_UNICODE[35504] := 16#E5E3;
   // GBK_TO_UNICODE[35505] := 16#9088;
   // GBK_TO_UNICODE[35506] := 16#E5E4;
   // GBK_TO_UNICODE[35507] := 16#9083;
   // GBK_TO_UNICODE[35508] := 16#E5E5;
   // GBK_TO_UNICODE[35509] := 16#908B;
   // GBK_TO_UNICODE[35510] := 16#E5E6;
   // GBK_TO_UNICODE[35511] := 16#5F50;
   // GBK_TO_UNICODE[35512] := 16#E5E7;
   // GBK_TO_UNICODE[35513] := 16#5F57;
   // GBK_TO_UNICODE[35514] := 16#E5E8;
   // GBK_TO_UNICODE[35515] := 16#5F56;
   // GBK_TO_UNICODE[35516] := 16#E5E9;
   // GBK_TO_UNICODE[35517] := 16#5F58;
   // GBK_TO_UNICODE[35518] := 16#E5EA;
   // GBK_TO_UNICODE[35519] := 16#5C3B;
   // GBK_TO_UNICODE[35520] := 16#E5EB;
   // GBK_TO_UNICODE[35521] := 16#54AB;
   // GBK_TO_UNICODE[35522] := 16#E5EC;
   // GBK_TO_UNICODE[35523] := 16#5C50;
   // GBK_TO_UNICODE[35524] := 16#E5ED;
   // GBK_TO_UNICODE[35525] := 16#5C59;
   // GBK_TO_UNICODE[35526] := 16#E5EE;
   // GBK_TO_UNICODE[35527] := 16#5B71;
   // GBK_TO_UNICODE[35528] := 16#E5EF;
   // GBK_TO_UNICODE[35529] := 16#5C63;
   // GBK_TO_UNICODE[35530] := 16#E5F0;
   // GBK_TO_UNICODE[35531] := 16#5C66;
   // GBK_TO_UNICODE[35532] := 16#E5F1;
   // GBK_TO_UNICODE[35533] := 16#7FBC;
   // GBK_TO_UNICODE[35534] := 16#E5F2;
   // GBK_TO_UNICODE[35535] := 16#5F2A;
   // GBK_TO_UNICODE[35536] := 16#E5F3;
   // GBK_TO_UNICODE[35537] := 16#5F29;
   // GBK_TO_UNICODE[35538] := 16#E5F4;
   // GBK_TO_UNICODE[35539] := 16#5F2D;
   // GBK_TO_UNICODE[35540] := 16#E5F5;
   // GBK_TO_UNICODE[35541] := 16#8274;
   // GBK_TO_UNICODE[35542] := 16#E5F6;
   // GBK_TO_UNICODE[35543] := 16#5F3C;
   // GBK_TO_UNICODE[35544] := 16#E5F7;
   // GBK_TO_UNICODE[35545] := 16#9B3B;
   // GBK_TO_UNICODE[35546] := 16#E5F8;
   // GBK_TO_UNICODE[35547] := 16#5C6E;
   // GBK_TO_UNICODE[35548] := 16#E5F9;
   // GBK_TO_UNICODE[35549] := 16#5981;
   // GBK_TO_UNICODE[35550] := 16#E5FA;
   // GBK_TO_UNICODE[35551] := 16#5983;
   // GBK_TO_UNICODE[35552] := 16#E5FB;
   // GBK_TO_UNICODE[35553] := 16#598D;
   // GBK_TO_UNICODE[35554] := 16#E5FC;
   // GBK_TO_UNICODE[35555] := 16#59A9;
   // GBK_TO_UNICODE[35556] := 16#E5FD;
   // GBK_TO_UNICODE[35557] := 16#59AA;
   // GBK_TO_UNICODE[35558] := 16#E5FE;
   // GBK_TO_UNICODE[35559] := 16#59A3;
   // GBK_TO_UNICODE[35560] := 16#E640;
   // GBK_TO_UNICODE[35561] := 16#936C;
   // GBK_TO_UNICODE[35562] := 16#E641;
   // GBK_TO_UNICODE[35563] := 16#936D;
   // GBK_TO_UNICODE[35564] := 16#E642;
   // GBK_TO_UNICODE[35565] := 16#936E;
   // GBK_TO_UNICODE[35566] := 16#E643;
   // GBK_TO_UNICODE[35567] := 16#936F;
   // GBK_TO_UNICODE[35568] := 16#E644;
   // GBK_TO_UNICODE[35569] := 16#9370;
   // GBK_TO_UNICODE[35570] := 16#E645;
   // GBK_TO_UNICODE[35571] := 16#9371;
   // GBK_TO_UNICODE[35572] := 16#E646;
   // GBK_TO_UNICODE[35573] := 16#9372;
   // GBK_TO_UNICODE[35574] := 16#E647;
   // GBK_TO_UNICODE[35575] := 16#9373;
   // GBK_TO_UNICODE[35576] := 16#E648;
   // GBK_TO_UNICODE[35577] := 16#9374;
   // GBK_TO_UNICODE[35578] := 16#E649;
   // GBK_TO_UNICODE[35579] := 16#9375;
   // GBK_TO_UNICODE[35580] := 16#E64A;
   // GBK_TO_UNICODE[35581] := 16#9376;
   // GBK_TO_UNICODE[35582] := 16#E64B;
   // GBK_TO_UNICODE[35583] := 16#9377;
   // GBK_TO_UNICODE[35584] := 16#E64C;
   // GBK_TO_UNICODE[35585] := 16#9378;
   // GBK_TO_UNICODE[35586] := 16#E64D;
   // GBK_TO_UNICODE[35587] := 16#9379;
   // GBK_TO_UNICODE[35588] := 16#E64E;
   // GBK_TO_UNICODE[35589] := 16#937A;
   // GBK_TO_UNICODE[35590] := 16#E64F;
   // GBK_TO_UNICODE[35591] := 16#937B;
   // GBK_TO_UNICODE[35592] := 16#E650;
   // GBK_TO_UNICODE[35593] := 16#937C;
   // GBK_TO_UNICODE[35594] := 16#E651;
   // GBK_TO_UNICODE[35595] := 16#937D;
   // GBK_TO_UNICODE[35596] := 16#E652;
   // GBK_TO_UNICODE[35597] := 16#937E;
   // GBK_TO_UNICODE[35598] := 16#E653;
   // GBK_TO_UNICODE[35599] := 16#937F;
   // GBK_TO_UNICODE[35600] := 16#E654;
   // GBK_TO_UNICODE[35601] := 16#9380;
   // GBK_TO_UNICODE[35602] := 16#E655;
   // GBK_TO_UNICODE[35603] := 16#9381;
   // GBK_TO_UNICODE[35604] := 16#E656;
   // GBK_TO_UNICODE[35605] := 16#9382;
   // GBK_TO_UNICODE[35606] := 16#E657;
   // GBK_TO_UNICODE[35607] := 16#9383;
   // GBK_TO_UNICODE[35608] := 16#E658;
   // GBK_TO_UNICODE[35609] := 16#9384;
   // GBK_TO_UNICODE[35610] := 16#E659;
   // GBK_TO_UNICODE[35611] := 16#9385;
   // GBK_TO_UNICODE[35612] := 16#E65A;
   // GBK_TO_UNICODE[35613] := 16#9386;
   // GBK_TO_UNICODE[35614] := 16#E65B;
   // GBK_TO_UNICODE[35615] := 16#9387;
   // GBK_TO_UNICODE[35616] := 16#E65C;
   // GBK_TO_UNICODE[35617] := 16#9388;
   // GBK_TO_UNICODE[35618] := 16#E65D;
   // GBK_TO_UNICODE[35619] := 16#9389;
   // GBK_TO_UNICODE[35620] := 16#E65E;
   // GBK_TO_UNICODE[35621] := 16#938A;
   // GBK_TO_UNICODE[35622] := 16#E65F;
   // GBK_TO_UNICODE[35623] := 16#938B;
   // GBK_TO_UNICODE[35624] := 16#E660;
   // GBK_TO_UNICODE[35625] := 16#938C;
   // GBK_TO_UNICODE[35626] := 16#E661;
   // GBK_TO_UNICODE[35627] := 16#938D;
   // GBK_TO_UNICODE[35628] := 16#E662;
   // GBK_TO_UNICODE[35629] := 16#938E;
   // GBK_TO_UNICODE[35630] := 16#E663;
   // GBK_TO_UNICODE[35631] := 16#9390;
   // GBK_TO_UNICODE[35632] := 16#E664;
   // GBK_TO_UNICODE[35633] := 16#9391;
   // GBK_TO_UNICODE[35634] := 16#E665;
   // GBK_TO_UNICODE[35635] := 16#9392;
   // GBK_TO_UNICODE[35636] := 16#E666;
   // GBK_TO_UNICODE[35637] := 16#9393;
   // GBK_TO_UNICODE[35638] := 16#E667;
   // GBK_TO_UNICODE[35639] := 16#9394;
   // GBK_TO_UNICODE[35640] := 16#E668;
   // GBK_TO_UNICODE[35641] := 16#9395;
   // GBK_TO_UNICODE[35642] := 16#E669;
   // GBK_TO_UNICODE[35643] := 16#9396;
   // GBK_TO_UNICODE[35644] := 16#E66A;
   // GBK_TO_UNICODE[35645] := 16#9397;
   // GBK_TO_UNICODE[35646] := 16#E66B;
   // GBK_TO_UNICODE[35647] := 16#9398;
   // GBK_TO_UNICODE[35648] := 16#E66C;
   // GBK_TO_UNICODE[35649] := 16#9399;
   // GBK_TO_UNICODE[35650] := 16#E66D;
   // GBK_TO_UNICODE[35651] := 16#939A;
   // GBK_TO_UNICODE[35652] := 16#E66E;
   // GBK_TO_UNICODE[35653] := 16#939B;
   // GBK_TO_UNICODE[35654] := 16#E66F;
   // GBK_TO_UNICODE[35655] := 16#939C;
   // GBK_TO_UNICODE[35656] := 16#E670;
   // GBK_TO_UNICODE[35657] := 16#939D;
   // GBK_TO_UNICODE[35658] := 16#E671;
   // GBK_TO_UNICODE[35659] := 16#939E;
   // GBK_TO_UNICODE[35660] := 16#E672;
   // GBK_TO_UNICODE[35661] := 16#939F;
   // GBK_TO_UNICODE[35662] := 16#E673;
   // GBK_TO_UNICODE[35663] := 16#93A0;
   // GBK_TO_UNICODE[35664] := 16#E674;
   // GBK_TO_UNICODE[35665] := 16#93A1;
   // GBK_TO_UNICODE[35666] := 16#E675;
   // GBK_TO_UNICODE[35667] := 16#93A2;
   // GBK_TO_UNICODE[35668] := 16#E676;
   // GBK_TO_UNICODE[35669] := 16#93A3;
   // GBK_TO_UNICODE[35670] := 16#E677;
   // GBK_TO_UNICODE[35671] := 16#93A4;
   // GBK_TO_UNICODE[35672] := 16#E678;
   // GBK_TO_UNICODE[35673] := 16#93A5;
   // GBK_TO_UNICODE[35674] := 16#E679;
   // GBK_TO_UNICODE[35675] := 16#93A6;
   // GBK_TO_UNICODE[35676] := 16#E67A;
   // GBK_TO_UNICODE[35677] := 16#93A7;
   // GBK_TO_UNICODE[35678] := 16#E67B;
   // GBK_TO_UNICODE[35679] := 16#93A8;
   // GBK_TO_UNICODE[35680] := 16#E67C;
   // GBK_TO_UNICODE[35681] := 16#93A9;
   // GBK_TO_UNICODE[35682] := 16#E67D;
   // GBK_TO_UNICODE[35683] := 16#93AA;
   // GBK_TO_UNICODE[35684] := 16#E67E;
   // GBK_TO_UNICODE[35685] := 16#93AB;
   // GBK_TO_UNICODE[35686] := 16#E680;
   // GBK_TO_UNICODE[35687] := 16#93AC;
   // GBK_TO_UNICODE[35688] := 16#E681;
   // GBK_TO_UNICODE[35689] := 16#93AD;
   // GBK_TO_UNICODE[35690] := 16#E682;
   // GBK_TO_UNICODE[35691] := 16#93AE;
   // GBK_TO_UNICODE[35692] := 16#E683;
   // GBK_TO_UNICODE[35693] := 16#93AF;
   // GBK_TO_UNICODE[35694] := 16#E684;
   // GBK_TO_UNICODE[35695] := 16#93B0;
   // GBK_TO_UNICODE[35696] := 16#E685;
   // GBK_TO_UNICODE[35697] := 16#93B1;
   // GBK_TO_UNICODE[35698] := 16#E686;
   // GBK_TO_UNICODE[35699] := 16#93B2;
   // GBK_TO_UNICODE[35700] := 16#E687;
   // GBK_TO_UNICODE[35701] := 16#93B3;
   // GBK_TO_UNICODE[35702] := 16#E688;
   // GBK_TO_UNICODE[35703] := 16#93B4;
   // GBK_TO_UNICODE[35704] := 16#E689;
   // GBK_TO_UNICODE[35705] := 16#93B5;
   // GBK_TO_UNICODE[35706] := 16#E68A;
   // GBK_TO_UNICODE[35707] := 16#93B6;
   // GBK_TO_UNICODE[35708] := 16#E68B;
   // GBK_TO_UNICODE[35709] := 16#93B7;
   // GBK_TO_UNICODE[35710] := 16#E68C;
   // GBK_TO_UNICODE[35711] := 16#93B8;
   // GBK_TO_UNICODE[35712] := 16#E68D;
   // GBK_TO_UNICODE[35713] := 16#93B9;
   // GBK_TO_UNICODE[35714] := 16#E68E;
   // GBK_TO_UNICODE[35715] := 16#93BA;
   // GBK_TO_UNICODE[35716] := 16#E68F;
   // GBK_TO_UNICODE[35717] := 16#93BB;
   // GBK_TO_UNICODE[35718] := 16#E690;
   // GBK_TO_UNICODE[35719] := 16#93BC;
   // GBK_TO_UNICODE[35720] := 16#E691;
   // GBK_TO_UNICODE[35721] := 16#93BD;
   // GBK_TO_UNICODE[35722] := 16#E692;
   // GBK_TO_UNICODE[35723] := 16#93BE;
   // GBK_TO_UNICODE[35724] := 16#E693;
   // GBK_TO_UNICODE[35725] := 16#93BF;
   // GBK_TO_UNICODE[35726] := 16#E694;
   // GBK_TO_UNICODE[35727] := 16#93C0;
   // GBK_TO_UNICODE[35728] := 16#E695;
   // GBK_TO_UNICODE[35729] := 16#93C1;
   // GBK_TO_UNICODE[35730] := 16#E696;
   // GBK_TO_UNICODE[35731] := 16#93C2;
   // GBK_TO_UNICODE[35732] := 16#E697;
   // GBK_TO_UNICODE[35733] := 16#93C3;
   // GBK_TO_UNICODE[35734] := 16#E698;
   // GBK_TO_UNICODE[35735] := 16#93C4;
   // GBK_TO_UNICODE[35736] := 16#E699;
   // GBK_TO_UNICODE[35737] := 16#93C5;
   // GBK_TO_UNICODE[35738] := 16#E69A;
   // GBK_TO_UNICODE[35739] := 16#93C6;
   // GBK_TO_UNICODE[35740] := 16#E69B;
   // GBK_TO_UNICODE[35741] := 16#93C7;
   // GBK_TO_UNICODE[35742] := 16#E69C;
   // GBK_TO_UNICODE[35743] := 16#93C8;
   // GBK_TO_UNICODE[35744] := 16#E69D;
   // GBK_TO_UNICODE[35745] := 16#93C9;
   // GBK_TO_UNICODE[35746] := 16#E69E;
   // GBK_TO_UNICODE[35747] := 16#93CB;
   // GBK_TO_UNICODE[35748] := 16#E69F;
   // GBK_TO_UNICODE[35749] := 16#93CC;
   // GBK_TO_UNICODE[35750] := 16#E6A0;
   // GBK_TO_UNICODE[35751] := 16#93CD;
   // GBK_TO_UNICODE[35752] := 16#E6A1;
   // GBK_TO_UNICODE[35753] := 16#5997;
   // GBK_TO_UNICODE[35754] := 16#E6A2;
   // GBK_TO_UNICODE[35755] := 16#59CA;
   // GBK_TO_UNICODE[35756] := 16#E6A3;
   // GBK_TO_UNICODE[35757] := 16#59AB;
   // GBK_TO_UNICODE[35758] := 16#E6A4;
   // GBK_TO_UNICODE[35759] := 16#599E;
   // GBK_TO_UNICODE[35760] := 16#E6A5;
   // GBK_TO_UNICODE[35761] := 16#59A4;
   // GBK_TO_UNICODE[35762] := 16#E6A6;
   // GBK_TO_UNICODE[35763] := 16#59D2;
   // GBK_TO_UNICODE[35764] := 16#E6A7;
   // GBK_TO_UNICODE[35765] := 16#59B2;
   // GBK_TO_UNICODE[35766] := 16#E6A8;
   // GBK_TO_UNICODE[35767] := 16#59AF;
   // GBK_TO_UNICODE[35768] := 16#E6A9;
   // GBK_TO_UNICODE[35769] := 16#59D7;
   // GBK_TO_UNICODE[35770] := 16#E6AA;
   // GBK_TO_UNICODE[35771] := 16#59BE;
   // GBK_TO_UNICODE[35772] := 16#E6AB;
   // GBK_TO_UNICODE[35773] := 16#5A05;
   // GBK_TO_UNICODE[35774] := 16#E6AC;
   // GBK_TO_UNICODE[35775] := 16#5A06;
   // GBK_TO_UNICODE[35776] := 16#E6AD;
   // GBK_TO_UNICODE[35777] := 16#59DD;
   // GBK_TO_UNICODE[35778] := 16#E6AE;
   // GBK_TO_UNICODE[35779] := 16#5A08;
   // GBK_TO_UNICODE[35780] := 16#E6AF;
   // GBK_TO_UNICODE[35781] := 16#59E3;
   // GBK_TO_UNICODE[35782] := 16#E6B0;
   // GBK_TO_UNICODE[35783] := 16#59D8;
   // GBK_TO_UNICODE[35784] := 16#E6B1;
   // GBK_TO_UNICODE[35785] := 16#59F9;
   // GBK_TO_UNICODE[35786] := 16#E6B2;
   // GBK_TO_UNICODE[35787] := 16#5A0C;
   // GBK_TO_UNICODE[35788] := 16#E6B3;
   // GBK_TO_UNICODE[35789] := 16#5A09;
   // GBK_TO_UNICODE[35790] := 16#E6B4;
   // GBK_TO_UNICODE[35791] := 16#5A32;
   // GBK_TO_UNICODE[35792] := 16#E6B5;
   // GBK_TO_UNICODE[35793] := 16#5A34;
   // GBK_TO_UNICODE[35794] := 16#E6B6;
   // GBK_TO_UNICODE[35795] := 16#5A11;
   // GBK_TO_UNICODE[35796] := 16#E6B7;
   // GBK_TO_UNICODE[35797] := 16#5A23;
   // GBK_TO_UNICODE[35798] := 16#E6B8;
   // GBK_TO_UNICODE[35799] := 16#5A13;
   // GBK_TO_UNICODE[35800] := 16#E6B9;
   // GBK_TO_UNICODE[35801] := 16#5A40;
   // GBK_TO_UNICODE[35802] := 16#E6BA;
   // GBK_TO_UNICODE[35803] := 16#5A67;
   // GBK_TO_UNICODE[35804] := 16#E6BB;
   // GBK_TO_UNICODE[35805] := 16#5A4A;
   // GBK_TO_UNICODE[35806] := 16#E6BC;
   // GBK_TO_UNICODE[35807] := 16#5A55;
   // GBK_TO_UNICODE[35808] := 16#E6BD;
   // GBK_TO_UNICODE[35809] := 16#5A3C;
   // GBK_TO_UNICODE[35810] := 16#E6BE;
   // GBK_TO_UNICODE[35811] := 16#5A62;
   // GBK_TO_UNICODE[35812] := 16#E6BF;
   // GBK_TO_UNICODE[35813] := 16#5A75;
   // GBK_TO_UNICODE[35814] := 16#E6C0;
   // GBK_TO_UNICODE[35815] := 16#80EC;
   // GBK_TO_UNICODE[35816] := 16#E6C1;
   // GBK_TO_UNICODE[35817] := 16#5AAA;
   // GBK_TO_UNICODE[35818] := 16#E6C2;
   // GBK_TO_UNICODE[35819] := 16#5A9B;
   // GBK_TO_UNICODE[35820] := 16#E6C3;
   // GBK_TO_UNICODE[35821] := 16#5A77;
   // GBK_TO_UNICODE[35822] := 16#E6C4;
   // GBK_TO_UNICODE[35823] := 16#5A7A;
   // GBK_TO_UNICODE[35824] := 16#E6C5;
   // GBK_TO_UNICODE[35825] := 16#5ABE;
   // GBK_TO_UNICODE[35826] := 16#E6C6;
   // GBK_TO_UNICODE[35827] := 16#5AEB;
   // GBK_TO_UNICODE[35828] := 16#E6C7;
   // GBK_TO_UNICODE[35829] := 16#5AB2;
   // GBK_TO_UNICODE[35830] := 16#E6C8;
   // GBK_TO_UNICODE[35831] := 16#5AD2;
   // GBK_TO_UNICODE[35832] := 16#E6C9;
   // GBK_TO_UNICODE[35833] := 16#5AD4;
   // GBK_TO_UNICODE[35834] := 16#E6CA;
   // GBK_TO_UNICODE[35835] := 16#5AB8;
   // GBK_TO_UNICODE[35836] := 16#E6CB;
   // GBK_TO_UNICODE[35837] := 16#5AE0;
   // GBK_TO_UNICODE[35838] := 16#E6CC;
   // GBK_TO_UNICODE[35839] := 16#5AE3;
   // GBK_TO_UNICODE[35840] := 16#E6CD;
   // GBK_TO_UNICODE[35841] := 16#5AF1;
   // GBK_TO_UNICODE[35842] := 16#E6CE;
   // GBK_TO_UNICODE[35843] := 16#5AD6;
   // GBK_TO_UNICODE[35844] := 16#E6CF;
   // GBK_TO_UNICODE[35845] := 16#5AE6;
   // GBK_TO_UNICODE[35846] := 16#E6D0;
   // GBK_TO_UNICODE[35847] := 16#5AD8;
   // GBK_TO_UNICODE[35848] := 16#E6D1;
   // GBK_TO_UNICODE[35849] := 16#5ADC;
   // GBK_TO_UNICODE[35850] := 16#E6D2;
   // GBK_TO_UNICODE[35851] := 16#5B09;
   // GBK_TO_UNICODE[35852] := 16#E6D3;
   // GBK_TO_UNICODE[35853] := 16#5B17;
   // GBK_TO_UNICODE[35854] := 16#E6D4;
   // GBK_TO_UNICODE[35855] := 16#5B16;
   // GBK_TO_UNICODE[35856] := 16#E6D5;
   // GBK_TO_UNICODE[35857] := 16#5B32;
   // GBK_TO_UNICODE[35858] := 16#E6D6;
   // GBK_TO_UNICODE[35859] := 16#5B37;
   // GBK_TO_UNICODE[35860] := 16#E6D7;
   // GBK_TO_UNICODE[35861] := 16#5B40;
   // GBK_TO_UNICODE[35862] := 16#E6D8;
   // GBK_TO_UNICODE[35863] := 16#5C15;
   // GBK_TO_UNICODE[35864] := 16#E6D9;
   // GBK_TO_UNICODE[35865] := 16#5C1C;
   // GBK_TO_UNICODE[35866] := 16#E6DA;
   // GBK_TO_UNICODE[35867] := 16#5B5A;
   // GBK_TO_UNICODE[35868] := 16#E6DB;
   // GBK_TO_UNICODE[35869] := 16#5B65;
   // GBK_TO_UNICODE[35870] := 16#E6DC;
   // GBK_TO_UNICODE[35871] := 16#5B73;
   // GBK_TO_UNICODE[35872] := 16#E6DD;
   // GBK_TO_UNICODE[35873] := 16#5B51;
   // GBK_TO_UNICODE[35874] := 16#E6DE;
   // GBK_TO_UNICODE[35875] := 16#5B53;
   // GBK_TO_UNICODE[35876] := 16#E6DF;
   // GBK_TO_UNICODE[35877] := 16#5B62;
   // GBK_TO_UNICODE[35878] := 16#E6E0;
   // GBK_TO_UNICODE[35879] := 16#9A75;
   // GBK_TO_UNICODE[35880] := 16#E6E1;
   // GBK_TO_UNICODE[35881] := 16#9A77;
   // GBK_TO_UNICODE[35882] := 16#E6E2;
   // GBK_TO_UNICODE[35883] := 16#9A78;
   // GBK_TO_UNICODE[35884] := 16#E6E3;
   // GBK_TO_UNICODE[35885] := 16#9A7A;
   // GBK_TO_UNICODE[35886] := 16#E6E4;
   // GBK_TO_UNICODE[35887] := 16#9A7F;
   // GBK_TO_UNICODE[35888] := 16#E6E5;
   // GBK_TO_UNICODE[35889] := 16#9A7D;
   // GBK_TO_UNICODE[35890] := 16#E6E6;
   // GBK_TO_UNICODE[35891] := 16#9A80;
   // GBK_TO_UNICODE[35892] := 16#E6E7;
   // GBK_TO_UNICODE[35893] := 16#9A81;
   // GBK_TO_UNICODE[35894] := 16#E6E8;
   // GBK_TO_UNICODE[35895] := 16#9A85;
   // GBK_TO_UNICODE[35896] := 16#E6E9;
   // GBK_TO_UNICODE[35897] := 16#9A88;
   // GBK_TO_UNICODE[35898] := 16#E6EA;
   // GBK_TO_UNICODE[35899] := 16#9A8A;
   // GBK_TO_UNICODE[35900] := 16#E6EB;
   // GBK_TO_UNICODE[35901] := 16#9A90;
   // GBK_TO_UNICODE[35902] := 16#E6EC;
   // GBK_TO_UNICODE[35903] := 16#9A92;
   // GBK_TO_UNICODE[35904] := 16#E6ED;
   // GBK_TO_UNICODE[35905] := 16#9A93;
   // GBK_TO_UNICODE[35906] := 16#E6EE;
   // GBK_TO_UNICODE[35907] := 16#9A96;
   // GBK_TO_UNICODE[35908] := 16#E6EF;
   // GBK_TO_UNICODE[35909] := 16#9A98;
   // GBK_TO_UNICODE[35910] := 16#E6F0;
   // GBK_TO_UNICODE[35911] := 16#9A9B;
   // GBK_TO_UNICODE[35912] := 16#E6F1;
   // GBK_TO_UNICODE[35913] := 16#9A9C;
   // GBK_TO_UNICODE[35914] := 16#E6F2;
   // GBK_TO_UNICODE[35915] := 16#9A9D;
   // GBK_TO_UNICODE[35916] := 16#E6F3;
   // GBK_TO_UNICODE[35917] := 16#9A9F;
   // GBK_TO_UNICODE[35918] := 16#E6F4;
   // GBK_TO_UNICODE[35919] := 16#9AA0;
   // GBK_TO_UNICODE[35920] := 16#E6F5;
   // GBK_TO_UNICODE[35921] := 16#9AA2;
   // GBK_TO_UNICODE[35922] := 16#E6F6;
   // GBK_TO_UNICODE[35923] := 16#9AA3;
   // GBK_TO_UNICODE[35924] := 16#E6F7;
   // GBK_TO_UNICODE[35925] := 16#9AA5;
   // GBK_TO_UNICODE[35926] := 16#E6F8;
   // GBK_TO_UNICODE[35927] := 16#9AA7;
   // GBK_TO_UNICODE[35928] := 16#E6F9;
   // GBK_TO_UNICODE[35929] := 16#7E9F;
   // GBK_TO_UNICODE[35930] := 16#E6FA;
   // GBK_TO_UNICODE[35931] := 16#7EA1;
   // GBK_TO_UNICODE[35932] := 16#E6FB;
   // GBK_TO_UNICODE[35933] := 16#7EA3;
   // GBK_TO_UNICODE[35934] := 16#E6FC;
   // GBK_TO_UNICODE[35935] := 16#7EA5;
   // GBK_TO_UNICODE[35936] := 16#E6FD;
   // GBK_TO_UNICODE[35937] := 16#7EA8;
   // GBK_TO_UNICODE[35938] := 16#E6FE;
   // GBK_TO_UNICODE[35939] := 16#7EA9;
   // GBK_TO_UNICODE[35940] := 16#E740;
   // GBK_TO_UNICODE[35941] := 16#93CE;
   // GBK_TO_UNICODE[35942] := 16#E741;
   // GBK_TO_UNICODE[35943] := 16#93CF;
   // GBK_TO_UNICODE[35944] := 16#E742;
   // GBK_TO_UNICODE[35945] := 16#93D0;
   // GBK_TO_UNICODE[35946] := 16#E743;
   // GBK_TO_UNICODE[35947] := 16#93D1;
   // GBK_TO_UNICODE[35948] := 16#E744;
   // GBK_TO_UNICODE[35949] := 16#93D2;
   // GBK_TO_UNICODE[35950] := 16#E745;
   // GBK_TO_UNICODE[35951] := 16#93D3;
   // GBK_TO_UNICODE[35952] := 16#E746;
   // GBK_TO_UNICODE[35953] := 16#93D4;
   // GBK_TO_UNICODE[35954] := 16#E747;
   // GBK_TO_UNICODE[35955] := 16#93D5;
   // GBK_TO_UNICODE[35956] := 16#E748;
   // GBK_TO_UNICODE[35957] := 16#93D7;
   // GBK_TO_UNICODE[35958] := 16#E749;
   // GBK_TO_UNICODE[35959] := 16#93D8;
   // GBK_TO_UNICODE[35960] := 16#E74A;
   // GBK_TO_UNICODE[35961] := 16#93D9;
   // GBK_TO_UNICODE[35962] := 16#E74B;
   // GBK_TO_UNICODE[35963] := 16#93DA;
   // GBK_TO_UNICODE[35964] := 16#E74C;
   // GBK_TO_UNICODE[35965] := 16#93DB;
   // GBK_TO_UNICODE[35966] := 16#E74D;
   // GBK_TO_UNICODE[35967] := 16#93DC;
   // GBK_TO_UNICODE[35968] := 16#E74E;
   // GBK_TO_UNICODE[35969] := 16#93DD;
   // GBK_TO_UNICODE[35970] := 16#E74F;
   // GBK_TO_UNICODE[35971] := 16#93DE;
   // GBK_TO_UNICODE[35972] := 16#E750;
   // GBK_TO_UNICODE[35973] := 16#93DF;
   // GBK_TO_UNICODE[35974] := 16#E751;
   // GBK_TO_UNICODE[35975] := 16#93E0;
   // GBK_TO_UNICODE[35976] := 16#E752;
   // GBK_TO_UNICODE[35977] := 16#93E1;
   // GBK_TO_UNICODE[35978] := 16#E753;
   // GBK_TO_UNICODE[35979] := 16#93E2;
   // GBK_TO_UNICODE[35980] := 16#E754;
   // GBK_TO_UNICODE[35981] := 16#93E3;
   // GBK_TO_UNICODE[35982] := 16#E755;
   // GBK_TO_UNICODE[35983] := 16#93E4;
   // GBK_TO_UNICODE[35984] := 16#E756;
   // GBK_TO_UNICODE[35985] := 16#93E5;
   // GBK_TO_UNICODE[35986] := 16#E757;
   // GBK_TO_UNICODE[35987] := 16#93E6;
   // GBK_TO_UNICODE[35988] := 16#E758;
   // GBK_TO_UNICODE[35989] := 16#93E7;
   // GBK_TO_UNICODE[35990] := 16#E759;
   // GBK_TO_UNICODE[35991] := 16#93E8;
   // GBK_TO_UNICODE[35992] := 16#E75A;
   // GBK_TO_UNICODE[35993] := 16#93E9;
   // GBK_TO_UNICODE[35994] := 16#E75B;
   // GBK_TO_UNICODE[35995] := 16#93EA;
   // GBK_TO_UNICODE[35996] := 16#E75C;
   // GBK_TO_UNICODE[35997] := 16#93EB;
   // GBK_TO_UNICODE[35998] := 16#E75D;
   // GBK_TO_UNICODE[35999] := 16#93EC;
   // GBK_TO_UNICODE[36000] := 16#E75E;
   // GBK_TO_UNICODE[36001] := 16#93ED;
   // GBK_TO_UNICODE[36002] := 16#E75F;
   // GBK_TO_UNICODE[36003] := 16#93EE;
   // GBK_TO_UNICODE[36004] := 16#E760;
   // GBK_TO_UNICODE[36005] := 16#93EF;
   // GBK_TO_UNICODE[36006] := 16#E761;
   // GBK_TO_UNICODE[36007] := 16#93F0;
   // GBK_TO_UNICODE[36008] := 16#E762;
   // GBK_TO_UNICODE[36009] := 16#93F1;
   // GBK_TO_UNICODE[36010] := 16#E763;
   // GBK_TO_UNICODE[36011] := 16#93F2;
   // GBK_TO_UNICODE[36012] := 16#E764;
   // GBK_TO_UNICODE[36013] := 16#93F3;
   // GBK_TO_UNICODE[36014] := 16#E765;
   // GBK_TO_UNICODE[36015] := 16#93F4;
   // GBK_TO_UNICODE[36016] := 16#E766;
   // GBK_TO_UNICODE[36017] := 16#93F5;
   // GBK_TO_UNICODE[36018] := 16#E767;
   // GBK_TO_UNICODE[36019] := 16#93F6;
   // GBK_TO_UNICODE[36020] := 16#E768;
   // GBK_TO_UNICODE[36021] := 16#93F7;
   // GBK_TO_UNICODE[36022] := 16#E769;
   // GBK_TO_UNICODE[36023] := 16#93F8;
   // GBK_TO_UNICODE[36024] := 16#E76A;
   // GBK_TO_UNICODE[36025] := 16#93F9;
   // GBK_TO_UNICODE[36026] := 16#E76B;
   // GBK_TO_UNICODE[36027] := 16#93FA;
   // GBK_TO_UNICODE[36028] := 16#E76C;
   // GBK_TO_UNICODE[36029] := 16#93FB;
   // GBK_TO_UNICODE[36030] := 16#E76D;
   // GBK_TO_UNICODE[36031] := 16#93FC;
   // GBK_TO_UNICODE[36032] := 16#E76E;
   // GBK_TO_UNICODE[36033] := 16#93FD;
   // GBK_TO_UNICODE[36034] := 16#E76F;
   // GBK_TO_UNICODE[36035] := 16#93FE;
   // GBK_TO_UNICODE[36036] := 16#E770;
   // GBK_TO_UNICODE[36037] := 16#93FF;
   // GBK_TO_UNICODE[36038] := 16#E771;
   // GBK_TO_UNICODE[36039] := 16#9400;
   // GBK_TO_UNICODE[36040] := 16#E772;
   // GBK_TO_UNICODE[36041] := 16#9401;
   // GBK_TO_UNICODE[36042] := 16#E773;
   // GBK_TO_UNICODE[36043] := 16#9402;
   // GBK_TO_UNICODE[36044] := 16#E774;
   // GBK_TO_UNICODE[36045] := 16#9403;
   // GBK_TO_UNICODE[36046] := 16#E775;
   // GBK_TO_UNICODE[36047] := 16#9404;
   // GBK_TO_UNICODE[36048] := 16#E776;
   // GBK_TO_UNICODE[36049] := 16#9405;
   // GBK_TO_UNICODE[36050] := 16#E777;
   // GBK_TO_UNICODE[36051] := 16#9406;
   // GBK_TO_UNICODE[36052] := 16#E778;
   // GBK_TO_UNICODE[36053] := 16#9407;
   // GBK_TO_UNICODE[36054] := 16#E779;
   // GBK_TO_UNICODE[36055] := 16#9408;
   // GBK_TO_UNICODE[36056] := 16#E77A;
   // GBK_TO_UNICODE[36057] := 16#9409;
   // GBK_TO_UNICODE[36058] := 16#E77B;
   // GBK_TO_UNICODE[36059] := 16#940A;
   // GBK_TO_UNICODE[36060] := 16#E77C;
   // GBK_TO_UNICODE[36061] := 16#940B;
   // GBK_TO_UNICODE[36062] := 16#E77D;
   // GBK_TO_UNICODE[36063] := 16#940C;
   // GBK_TO_UNICODE[36064] := 16#E77E;
   // GBK_TO_UNICODE[36065] := 16#940D;
   // GBK_TO_UNICODE[36066] := 16#E780;
   // GBK_TO_UNICODE[36067] := 16#940E;
   // GBK_TO_UNICODE[36068] := 16#E781;
   // GBK_TO_UNICODE[36069] := 16#940F;
   // GBK_TO_UNICODE[36070] := 16#E782;
   // GBK_TO_UNICODE[36071] := 16#9410;
   // GBK_TO_UNICODE[36072] := 16#E783;
   // GBK_TO_UNICODE[36073] := 16#9411;
   // GBK_TO_UNICODE[36074] := 16#E784;
   // GBK_TO_UNICODE[36075] := 16#9412;
   // GBK_TO_UNICODE[36076] := 16#E785;
   // GBK_TO_UNICODE[36077] := 16#9413;
   // GBK_TO_UNICODE[36078] := 16#E786;
   // GBK_TO_UNICODE[36079] := 16#9414;
   // GBK_TO_UNICODE[36080] := 16#E787;
   // GBK_TO_UNICODE[36081] := 16#9415;
   // GBK_TO_UNICODE[36082] := 16#E788;
   // GBK_TO_UNICODE[36083] := 16#9416;
   // GBK_TO_UNICODE[36084] := 16#E789;
   // GBK_TO_UNICODE[36085] := 16#9417;
   // GBK_TO_UNICODE[36086] := 16#E78A;
   // GBK_TO_UNICODE[36087] := 16#9418;
   // GBK_TO_UNICODE[36088] := 16#E78B;
   // GBK_TO_UNICODE[36089] := 16#9419;
   // GBK_TO_UNICODE[36090] := 16#E78C;
   // GBK_TO_UNICODE[36091] := 16#941A;
   // GBK_TO_UNICODE[36092] := 16#E78D;
   // GBK_TO_UNICODE[36093] := 16#941B;
   // GBK_TO_UNICODE[36094] := 16#E78E;
   // GBK_TO_UNICODE[36095] := 16#941C;
   // GBK_TO_UNICODE[36096] := 16#E78F;
   // GBK_TO_UNICODE[36097] := 16#941D;
   // GBK_TO_UNICODE[36098] := 16#E790;
   // GBK_TO_UNICODE[36099] := 16#941E;
   // GBK_TO_UNICODE[36100] := 16#E791;
   // GBK_TO_UNICODE[36101] := 16#941F;
   // GBK_TO_UNICODE[36102] := 16#E792;
   // GBK_TO_UNICODE[36103] := 16#9420;
   // GBK_TO_UNICODE[36104] := 16#E793;
   // GBK_TO_UNICODE[36105] := 16#9421;
   // GBK_TO_UNICODE[36106] := 16#E794;
   // GBK_TO_UNICODE[36107] := 16#9422;
   // GBK_TO_UNICODE[36108] := 16#E795;
   // GBK_TO_UNICODE[36109] := 16#9423;
   // GBK_TO_UNICODE[36110] := 16#E796;
   // GBK_TO_UNICODE[36111] := 16#9424;
   // GBK_TO_UNICODE[36112] := 16#E797;
   // GBK_TO_UNICODE[36113] := 16#9425;
   // GBK_TO_UNICODE[36114] := 16#E798;
   // GBK_TO_UNICODE[36115] := 16#9426;
   // GBK_TO_UNICODE[36116] := 16#E799;
   // GBK_TO_UNICODE[36117] := 16#9427;
   // GBK_TO_UNICODE[36118] := 16#E79A;
   // GBK_TO_UNICODE[36119] := 16#9428;
   // GBK_TO_UNICODE[36120] := 16#E79B;
   // GBK_TO_UNICODE[36121] := 16#9429;
   // GBK_TO_UNICODE[36122] := 16#E79C;
   // GBK_TO_UNICODE[36123] := 16#942A;
   // GBK_TO_UNICODE[36124] := 16#E79D;
   // GBK_TO_UNICODE[36125] := 16#942B;
   // GBK_TO_UNICODE[36126] := 16#E79E;
   // GBK_TO_UNICODE[36127] := 16#942C;
   // GBK_TO_UNICODE[36128] := 16#E79F;
   // GBK_TO_UNICODE[36129] := 16#942D;
   // GBK_TO_UNICODE[36130] := 16#E7A0;
   // GBK_TO_UNICODE[36131] := 16#942E;
   // GBK_TO_UNICODE[36132] := 16#E7A1;
   // GBK_TO_UNICODE[36133] := 16#7EAD;
   // GBK_TO_UNICODE[36134] := 16#E7A2;
   // GBK_TO_UNICODE[36135] := 16#7EB0;
   // GBK_TO_UNICODE[36136] := 16#E7A3;
   // GBK_TO_UNICODE[36137] := 16#7EBE;
   // GBK_TO_UNICODE[36138] := 16#E7A4;
   // GBK_TO_UNICODE[36139] := 16#7EC0;
   // GBK_TO_UNICODE[36140] := 16#E7A5;
   // GBK_TO_UNICODE[36141] := 16#7EC1;
   // GBK_TO_UNICODE[36142] := 16#E7A6;
   // GBK_TO_UNICODE[36143] := 16#7EC2;
   // GBK_TO_UNICODE[36144] := 16#E7A7;
   // GBK_TO_UNICODE[36145] := 16#7EC9;
   // GBK_TO_UNICODE[36146] := 16#E7A8;
   // GBK_TO_UNICODE[36147] := 16#7ECB;
   // GBK_TO_UNICODE[36148] := 16#E7A9;
   // GBK_TO_UNICODE[36149] := 16#7ECC;
   // GBK_TO_UNICODE[36150] := 16#E7AA;
   // GBK_TO_UNICODE[36151] := 16#7ED0;
   // GBK_TO_UNICODE[36152] := 16#E7AB;
   // GBK_TO_UNICODE[36153] := 16#7ED4;
   // GBK_TO_UNICODE[36154] := 16#E7AC;
   // GBK_TO_UNICODE[36155] := 16#7ED7;
   // GBK_TO_UNICODE[36156] := 16#E7AD;
   // GBK_TO_UNICODE[36157] := 16#7EDB;
   // GBK_TO_UNICODE[36158] := 16#E7AE;
   // GBK_TO_UNICODE[36159] := 16#7EE0;
   // GBK_TO_UNICODE[36160] := 16#E7AF;
   // GBK_TO_UNICODE[36161] := 16#7EE1;
   // GBK_TO_UNICODE[36162] := 16#E7B0;
   // GBK_TO_UNICODE[36163] := 16#7EE8;
   // GBK_TO_UNICODE[36164] := 16#E7B1;
   // GBK_TO_UNICODE[36165] := 16#7EEB;
   // GBK_TO_UNICODE[36166] := 16#E7B2;
   // GBK_TO_UNICODE[36167] := 16#7EEE;
   // GBK_TO_UNICODE[36168] := 16#E7B3;
   // GBK_TO_UNICODE[36169] := 16#7EEF;
   // GBK_TO_UNICODE[36170] := 16#E7B4;
   // GBK_TO_UNICODE[36171] := 16#7EF1;
   // GBK_TO_UNICODE[36172] := 16#E7B5;
   // GBK_TO_UNICODE[36173] := 16#7EF2;
   // GBK_TO_UNICODE[36174] := 16#E7B6;
   // GBK_TO_UNICODE[36175] := 16#7F0D;
   // GBK_TO_UNICODE[36176] := 16#E7B7;
   // GBK_TO_UNICODE[36177] := 16#7EF6;
   // GBK_TO_UNICODE[36178] := 16#E7B8;
   // GBK_TO_UNICODE[36179] := 16#7EFA;
   // GBK_TO_UNICODE[36180] := 16#E7B9;
   // GBK_TO_UNICODE[36181] := 16#7EFB;
   // GBK_TO_UNICODE[36182] := 16#E7BA;
   // GBK_TO_UNICODE[36183] := 16#7EFE;
   // GBK_TO_UNICODE[36184] := 16#E7BB;
   // GBK_TO_UNICODE[36185] := 16#7F01;
   // GBK_TO_UNICODE[36186] := 16#E7BC;
   // GBK_TO_UNICODE[36187] := 16#7F02;
   // GBK_TO_UNICODE[36188] := 16#E7BD;
   // GBK_TO_UNICODE[36189] := 16#7F03;
   // GBK_TO_UNICODE[36190] := 16#E7BE;
   // GBK_TO_UNICODE[36191] := 16#7F07;
   // GBK_TO_UNICODE[36192] := 16#E7BF;
   // GBK_TO_UNICODE[36193] := 16#7F08;
   // GBK_TO_UNICODE[36194] := 16#E7C0;
   // GBK_TO_UNICODE[36195] := 16#7F0B;
   // GBK_TO_UNICODE[36196] := 16#E7C1;
   // GBK_TO_UNICODE[36197] := 16#7F0C;
   // GBK_TO_UNICODE[36198] := 16#E7C2;
   // GBK_TO_UNICODE[36199] := 16#7F0F;
   // GBK_TO_UNICODE[36200] := 16#E7C3;
   // GBK_TO_UNICODE[36201] := 16#7F11;
   // GBK_TO_UNICODE[36202] := 16#E7C4;
   // GBK_TO_UNICODE[36203] := 16#7F12;
   // GBK_TO_UNICODE[36204] := 16#E7C5;
   // GBK_TO_UNICODE[36205] := 16#7F17;
   // GBK_TO_UNICODE[36206] := 16#E7C6;
   // GBK_TO_UNICODE[36207] := 16#7F19;
   // GBK_TO_UNICODE[36208] := 16#E7C7;
   // GBK_TO_UNICODE[36209] := 16#7F1C;
   // GBK_TO_UNICODE[36210] := 16#E7C8;
   // GBK_TO_UNICODE[36211] := 16#7F1B;
   // GBK_TO_UNICODE[36212] := 16#E7C9;
   // GBK_TO_UNICODE[36213] := 16#7F1F;
   // GBK_TO_UNICODE[36214] := 16#E7CA;
   // GBK_TO_UNICODE[36215] := 16#7F21;
   // GBK_TO_UNICODE[36216] := 16#E7CB;
   // GBK_TO_UNICODE[36217] := 16#7F22;
   // GBK_TO_UNICODE[36218] := 16#E7CC;
   // GBK_TO_UNICODE[36219] := 16#7F23;
   // GBK_TO_UNICODE[36220] := 16#E7CD;
   // GBK_TO_UNICODE[36221] := 16#7F24;
   // GBK_TO_UNICODE[36222] := 16#E7CE;
   // GBK_TO_UNICODE[36223] := 16#7F25;
   // GBK_TO_UNICODE[36224] := 16#E7CF;
   // GBK_TO_UNICODE[36225] := 16#7F26;
   // GBK_TO_UNICODE[36226] := 16#E7D0;
   // GBK_TO_UNICODE[36227] := 16#7F27;
   // GBK_TO_UNICODE[36228] := 16#E7D1;
   // GBK_TO_UNICODE[36229] := 16#7F2A;
   // GBK_TO_UNICODE[36230] := 16#E7D2;
   // GBK_TO_UNICODE[36231] := 16#7F2B;
   // GBK_TO_UNICODE[36232] := 16#E7D3;
   // GBK_TO_UNICODE[36233] := 16#7F2C;
   // GBK_TO_UNICODE[36234] := 16#E7D4;
   // GBK_TO_UNICODE[36235] := 16#7F2D;
   // GBK_TO_UNICODE[36236] := 16#E7D5;
   // GBK_TO_UNICODE[36237] := 16#7F2F;
   // GBK_TO_UNICODE[36238] := 16#E7D6;
   // GBK_TO_UNICODE[36239] := 16#7F30;
   // GBK_TO_UNICODE[36240] := 16#E7D7;
   // GBK_TO_UNICODE[36241] := 16#7F31;
   // GBK_TO_UNICODE[36242] := 16#E7D8;
   // GBK_TO_UNICODE[36243] := 16#7F32;
   // GBK_TO_UNICODE[36244] := 16#E7D9;
   // GBK_TO_UNICODE[36245] := 16#7F33;
   // GBK_TO_UNICODE[36246] := 16#E7DA;
   // GBK_TO_UNICODE[36247] := 16#7F35;
   // GBK_TO_UNICODE[36248] := 16#E7DB;
   // GBK_TO_UNICODE[36249] := 16#5E7A;
   // GBK_TO_UNICODE[36250] := 16#E7DC;
   // GBK_TO_UNICODE[36251] := 16#757F;
   // GBK_TO_UNICODE[36252] := 16#E7DD;
   // GBK_TO_UNICODE[36253] := 16#5DDB;
   // GBK_TO_UNICODE[36254] := 16#E7DE;
   // GBK_TO_UNICODE[36255] := 16#753E;
   // GBK_TO_UNICODE[36256] := 16#E7DF;
   // GBK_TO_UNICODE[36257] := 16#9095;
   // GBK_TO_UNICODE[36258] := 16#E7E0;
   // GBK_TO_UNICODE[36259] := 16#738E;
   // GBK_TO_UNICODE[36260] := 16#E7E1;
   // GBK_TO_UNICODE[36261] := 16#7391;
   // GBK_TO_UNICODE[36262] := 16#E7E2;
   // GBK_TO_UNICODE[36263] := 16#73AE;
   // GBK_TO_UNICODE[36264] := 16#E7E3;
   // GBK_TO_UNICODE[36265] := 16#73A2;
   // GBK_TO_UNICODE[36266] := 16#E7E4;
   // GBK_TO_UNICODE[36267] := 16#739F;
   // GBK_TO_UNICODE[36268] := 16#E7E5;
   // GBK_TO_UNICODE[36269] := 16#73CF;
   // GBK_TO_UNICODE[36270] := 16#E7E6;
   // GBK_TO_UNICODE[36271] := 16#73C2;
   // GBK_TO_UNICODE[36272] := 16#E7E7;
   // GBK_TO_UNICODE[36273] := 16#73D1;
   // GBK_TO_UNICODE[36274] := 16#E7E8;
   // GBK_TO_UNICODE[36275] := 16#73B7;
   // GBK_TO_UNICODE[36276] := 16#E7E9;
   // GBK_TO_UNICODE[36277] := 16#73B3;
   // GBK_TO_UNICODE[36278] := 16#E7EA;
   // GBK_TO_UNICODE[36279] := 16#73C0;
   // GBK_TO_UNICODE[36280] := 16#E7EB;
   // GBK_TO_UNICODE[36281] := 16#73C9;
   // GBK_TO_UNICODE[36282] := 16#E7EC;
   // GBK_TO_UNICODE[36283] := 16#73C8;
   // GBK_TO_UNICODE[36284] := 16#E7ED;
   // GBK_TO_UNICODE[36285] := 16#73E5;
   // GBK_TO_UNICODE[36286] := 16#E7EE;
   // GBK_TO_UNICODE[36287] := 16#73D9;
   // GBK_TO_UNICODE[36288] := 16#E7EF;
   // GBK_TO_UNICODE[36289] := 16#987C;
   // GBK_TO_UNICODE[36290] := 16#E7F0;
   // GBK_TO_UNICODE[36291] := 16#740A;
   // GBK_TO_UNICODE[36292] := 16#E7F1;
   // GBK_TO_UNICODE[36293] := 16#73E9;
   // GBK_TO_UNICODE[36294] := 16#E7F2;
   // GBK_TO_UNICODE[36295] := 16#73E7;
   // GBK_TO_UNICODE[36296] := 16#E7F3;
   // GBK_TO_UNICODE[36297] := 16#73DE;
   // GBK_TO_UNICODE[36298] := 16#E7F4;
   // GBK_TO_UNICODE[36299] := 16#73BA;
   // GBK_TO_UNICODE[36300] := 16#E7F5;
   // GBK_TO_UNICODE[36301] := 16#73F2;
   // GBK_TO_UNICODE[36302] := 16#E7F6;
   // GBK_TO_UNICODE[36303] := 16#740F;
   // GBK_TO_UNICODE[36304] := 16#E7F7;
   // GBK_TO_UNICODE[36305] := 16#742A;
   // GBK_TO_UNICODE[36306] := 16#E7F8;
   // GBK_TO_UNICODE[36307] := 16#745B;
   // GBK_TO_UNICODE[36308] := 16#E7F9;
   // GBK_TO_UNICODE[36309] := 16#7426;
   // GBK_TO_UNICODE[36310] := 16#E7FA;
   // GBK_TO_UNICODE[36311] := 16#7425;
   // GBK_TO_UNICODE[36312] := 16#E7FB;
   // GBK_TO_UNICODE[36313] := 16#7428;
   // GBK_TO_UNICODE[36314] := 16#E7FC;
   // GBK_TO_UNICODE[36315] := 16#7430;
   // GBK_TO_UNICODE[36316] := 16#E7FD;
   // GBK_TO_UNICODE[36317] := 16#742E;
   // GBK_TO_UNICODE[36318] := 16#E7FE;
   // GBK_TO_UNICODE[36319] := 16#742C;
   // GBK_TO_UNICODE[36320] := 16#E840;
   // GBK_TO_UNICODE[36321] := 16#942F;
   // GBK_TO_UNICODE[36322] := 16#E841;
   // GBK_TO_UNICODE[36323] := 16#9430;
   // GBK_TO_UNICODE[36324] := 16#E842;
   // GBK_TO_UNICODE[36325] := 16#9431;
   // GBK_TO_UNICODE[36326] := 16#E843;
   // GBK_TO_UNICODE[36327] := 16#9432;
   // GBK_TO_UNICODE[36328] := 16#E844;
   // GBK_TO_UNICODE[36329] := 16#9433;
   // GBK_TO_UNICODE[36330] := 16#E845;
   // GBK_TO_UNICODE[36331] := 16#9434;
   // GBK_TO_UNICODE[36332] := 16#E846;
   // GBK_TO_UNICODE[36333] := 16#9435;
   // GBK_TO_UNICODE[36334] := 16#E847;
   // GBK_TO_UNICODE[36335] := 16#9436;
   // GBK_TO_UNICODE[36336] := 16#E848;
   // GBK_TO_UNICODE[36337] := 16#9437;
   // GBK_TO_UNICODE[36338] := 16#E849;
   // GBK_TO_UNICODE[36339] := 16#9438;
   // GBK_TO_UNICODE[36340] := 16#E84A;
   // GBK_TO_UNICODE[36341] := 16#9439;
   // GBK_TO_UNICODE[36342] := 16#E84B;
   // GBK_TO_UNICODE[36343] := 16#943A;
   // GBK_TO_UNICODE[36344] := 16#E84C;
   // GBK_TO_UNICODE[36345] := 16#943B;
   // GBK_TO_UNICODE[36346] := 16#E84D;
   // GBK_TO_UNICODE[36347] := 16#943C;
   // GBK_TO_UNICODE[36348] := 16#E84E;
   // GBK_TO_UNICODE[36349] := 16#943D;
   // GBK_TO_UNICODE[36350] := 16#E84F;
   // GBK_TO_UNICODE[36351] := 16#943F;
   // GBK_TO_UNICODE[36352] := 16#E850;
   // GBK_TO_UNICODE[36353] := 16#9440;
   // GBK_TO_UNICODE[36354] := 16#E851;
   // GBK_TO_UNICODE[36355] := 16#9441;
   // GBK_TO_UNICODE[36356] := 16#E852;
   // GBK_TO_UNICODE[36357] := 16#9442;
   // GBK_TO_UNICODE[36358] := 16#E853;
   // GBK_TO_UNICODE[36359] := 16#9443;
   // GBK_TO_UNICODE[36360] := 16#E854;
   // GBK_TO_UNICODE[36361] := 16#9444;
   // GBK_TO_UNICODE[36362] := 16#E855;
   // GBK_TO_UNICODE[36363] := 16#9445;
   // GBK_TO_UNICODE[36364] := 16#E856;
   // GBK_TO_UNICODE[36365] := 16#9446;
   // GBK_TO_UNICODE[36366] := 16#E857;
   // GBK_TO_UNICODE[36367] := 16#9447;
   // GBK_TO_UNICODE[36368] := 16#E858;
   // GBK_TO_UNICODE[36369] := 16#9448;
   // GBK_TO_UNICODE[36370] := 16#E859;
   // GBK_TO_UNICODE[36371] := 16#9449;
   // GBK_TO_UNICODE[36372] := 16#E85A;
   // GBK_TO_UNICODE[36373] := 16#944A;
   // GBK_TO_UNICODE[36374] := 16#E85B;
   // GBK_TO_UNICODE[36375] := 16#944B;
   // GBK_TO_UNICODE[36376] := 16#E85C;
   // GBK_TO_UNICODE[36377] := 16#944C;
   // GBK_TO_UNICODE[36378] := 16#E85D;
   // GBK_TO_UNICODE[36379] := 16#944D;
   // GBK_TO_UNICODE[36380] := 16#E85E;
   // GBK_TO_UNICODE[36381] := 16#944E;
   // GBK_TO_UNICODE[36382] := 16#E85F;
   // GBK_TO_UNICODE[36383] := 16#944F;
   // GBK_TO_UNICODE[36384] := 16#E860;
   // GBK_TO_UNICODE[36385] := 16#9450;
   // GBK_TO_UNICODE[36386] := 16#E861;
   // GBK_TO_UNICODE[36387] := 16#9451;
   // GBK_TO_UNICODE[36388] := 16#E862;
   // GBK_TO_UNICODE[36389] := 16#9452;
   // GBK_TO_UNICODE[36390] := 16#E863;
   // GBK_TO_UNICODE[36391] := 16#9453;
   // GBK_TO_UNICODE[36392] := 16#E864;
   // GBK_TO_UNICODE[36393] := 16#9454;
   // GBK_TO_UNICODE[36394] := 16#E865;
   // GBK_TO_UNICODE[36395] := 16#9455;
   // GBK_TO_UNICODE[36396] := 16#E866;
   // GBK_TO_UNICODE[36397] := 16#9456;
   // GBK_TO_UNICODE[36398] := 16#E867;
   // GBK_TO_UNICODE[36399] := 16#9457;
   // GBK_TO_UNICODE[36400] := 16#E868;
   // GBK_TO_UNICODE[36401] := 16#9458;
   // GBK_TO_UNICODE[36402] := 16#E869;
   // GBK_TO_UNICODE[36403] := 16#9459;
   // GBK_TO_UNICODE[36404] := 16#E86A;
   // GBK_TO_UNICODE[36405] := 16#945A;
   // GBK_TO_UNICODE[36406] := 16#E86B;
   // GBK_TO_UNICODE[36407] := 16#945B;
   // GBK_TO_UNICODE[36408] := 16#E86C;
   // GBK_TO_UNICODE[36409] := 16#945C;
   // GBK_TO_UNICODE[36410] := 16#E86D;
   // GBK_TO_UNICODE[36411] := 16#945D;
   // GBK_TO_UNICODE[36412] := 16#E86E;
   // GBK_TO_UNICODE[36413] := 16#945E;
   // GBK_TO_UNICODE[36414] := 16#E86F;
   // GBK_TO_UNICODE[36415] := 16#945F;
   // GBK_TO_UNICODE[36416] := 16#E870;
   // GBK_TO_UNICODE[36417] := 16#9460;
   // GBK_TO_UNICODE[36418] := 16#E871;
   // GBK_TO_UNICODE[36419] := 16#9461;
   // GBK_TO_UNICODE[36420] := 16#E872;
   // GBK_TO_UNICODE[36421] := 16#9462;
   // GBK_TO_UNICODE[36422] := 16#E873;
   // GBK_TO_UNICODE[36423] := 16#9463;
   // GBK_TO_UNICODE[36424] := 16#E874;
   // GBK_TO_UNICODE[36425] := 16#9464;
   // GBK_TO_UNICODE[36426] := 16#E875;
   // GBK_TO_UNICODE[36427] := 16#9465;
   // GBK_TO_UNICODE[36428] := 16#E876;
   // GBK_TO_UNICODE[36429] := 16#9466;
   // GBK_TO_UNICODE[36430] := 16#E877;
   // GBK_TO_UNICODE[36431] := 16#9467;
   // GBK_TO_UNICODE[36432] := 16#E878;
   // GBK_TO_UNICODE[36433] := 16#9468;
   // GBK_TO_UNICODE[36434] := 16#E879;
   // GBK_TO_UNICODE[36435] := 16#9469;
   // GBK_TO_UNICODE[36436] := 16#E87A;
   // GBK_TO_UNICODE[36437] := 16#946A;
   // GBK_TO_UNICODE[36438] := 16#E87B;
   // GBK_TO_UNICODE[36439] := 16#946C;
   // GBK_TO_UNICODE[36440] := 16#E87C;
   // GBK_TO_UNICODE[36441] := 16#946D;
   // GBK_TO_UNICODE[36442] := 16#E87D;
   // GBK_TO_UNICODE[36443] := 16#946E;
   // GBK_TO_UNICODE[36444] := 16#E87E;
   // GBK_TO_UNICODE[36445] := 16#946F;
   // GBK_TO_UNICODE[36446] := 16#E880;
   // GBK_TO_UNICODE[36447] := 16#9470;
   // GBK_TO_UNICODE[36448] := 16#E881;
   // GBK_TO_UNICODE[36449] := 16#9471;
   // GBK_TO_UNICODE[36450] := 16#E882;
   // GBK_TO_UNICODE[36451] := 16#9472;
   // GBK_TO_UNICODE[36452] := 16#E883;
   // GBK_TO_UNICODE[36453] := 16#9473;
   // GBK_TO_UNICODE[36454] := 16#E884;
   // GBK_TO_UNICODE[36455] := 16#9474;
   // GBK_TO_UNICODE[36456] := 16#E885;
   // GBK_TO_UNICODE[36457] := 16#9475;
   // GBK_TO_UNICODE[36458] := 16#E886;
   // GBK_TO_UNICODE[36459] := 16#9476;
   // GBK_TO_UNICODE[36460] := 16#E887;
   // GBK_TO_UNICODE[36461] := 16#9477;
   // GBK_TO_UNICODE[36462] := 16#E888;
   // GBK_TO_UNICODE[36463] := 16#9478;
   // GBK_TO_UNICODE[36464] := 16#E889;
   // GBK_TO_UNICODE[36465] := 16#9479;
   // GBK_TO_UNICODE[36466] := 16#E88A;
   // GBK_TO_UNICODE[36467] := 16#947A;
   // GBK_TO_UNICODE[36468] := 16#E88B;
   // GBK_TO_UNICODE[36469] := 16#947B;
   // GBK_TO_UNICODE[36470] := 16#E88C;
   // GBK_TO_UNICODE[36471] := 16#947C;
   // GBK_TO_UNICODE[36472] := 16#E88D;
   // GBK_TO_UNICODE[36473] := 16#947D;
   // GBK_TO_UNICODE[36474] := 16#E88E;
   // GBK_TO_UNICODE[36475] := 16#947E;
   // GBK_TO_UNICODE[36476] := 16#E88F;
   // GBK_TO_UNICODE[36477] := 16#947F;
   // GBK_TO_UNICODE[36478] := 16#E890;
   // GBK_TO_UNICODE[36479] := 16#9480;
   // GBK_TO_UNICODE[36480] := 16#E891;
   // GBK_TO_UNICODE[36481] := 16#9481;
   // GBK_TO_UNICODE[36482] := 16#E892;
   // GBK_TO_UNICODE[36483] := 16#9482;
   // GBK_TO_UNICODE[36484] := 16#E893;
   // GBK_TO_UNICODE[36485] := 16#9483;
   // GBK_TO_UNICODE[36486] := 16#E894;
   // GBK_TO_UNICODE[36487] := 16#9484;
   // GBK_TO_UNICODE[36488] := 16#E895;
   // GBK_TO_UNICODE[36489] := 16#9491;
   // GBK_TO_UNICODE[36490] := 16#E896;
   // GBK_TO_UNICODE[36491] := 16#9496;
   // GBK_TO_UNICODE[36492] := 16#E897;
   // GBK_TO_UNICODE[36493] := 16#9498;
   // GBK_TO_UNICODE[36494] := 16#E898;
   // GBK_TO_UNICODE[36495] := 16#94C7;
   // GBK_TO_UNICODE[36496] := 16#E899;
   // GBK_TO_UNICODE[36497] := 16#94CF;
   // GBK_TO_UNICODE[36498] := 16#E89A;
   // GBK_TO_UNICODE[36499] := 16#94D3;
   // GBK_TO_UNICODE[36500] := 16#E89B;
   // GBK_TO_UNICODE[36501] := 16#94D4;
   // GBK_TO_UNICODE[36502] := 16#E89C;
   // GBK_TO_UNICODE[36503] := 16#94DA;
   // GBK_TO_UNICODE[36504] := 16#E89D;
   // GBK_TO_UNICODE[36505] := 16#94E6;
   // GBK_TO_UNICODE[36506] := 16#E89E;
   // GBK_TO_UNICODE[36507] := 16#94FB;
   // GBK_TO_UNICODE[36508] := 16#E89F;
   // GBK_TO_UNICODE[36509] := 16#951C;
   // GBK_TO_UNICODE[36510] := 16#E8A0;
   // GBK_TO_UNICODE[36511] := 16#9520;
   // GBK_TO_UNICODE[36512] := 16#E8A1;
   // GBK_TO_UNICODE[36513] := 16#741B;
   // GBK_TO_UNICODE[36514] := 16#E8A2;
   // GBK_TO_UNICODE[36515] := 16#741A;
   // GBK_TO_UNICODE[36516] := 16#E8A3;
   // GBK_TO_UNICODE[36517] := 16#7441;
   // GBK_TO_UNICODE[36518] := 16#E8A4;
   // GBK_TO_UNICODE[36519] := 16#745C;
   // GBK_TO_UNICODE[36520] := 16#E8A5;
   // GBK_TO_UNICODE[36521] := 16#7457;
   // GBK_TO_UNICODE[36522] := 16#E8A6;
   // GBK_TO_UNICODE[36523] := 16#7455;
   // GBK_TO_UNICODE[36524] := 16#E8A7;
   // GBK_TO_UNICODE[36525] := 16#7459;
   // GBK_TO_UNICODE[36526] := 16#E8A8;
   // GBK_TO_UNICODE[36527] := 16#7477;
   // GBK_TO_UNICODE[36528] := 16#E8A9;
   // GBK_TO_UNICODE[36529] := 16#746D;
   // GBK_TO_UNICODE[36530] := 16#E8AA;
   // GBK_TO_UNICODE[36531] := 16#747E;
   // GBK_TO_UNICODE[36532] := 16#E8AB;
   // GBK_TO_UNICODE[36533] := 16#749C;
   // GBK_TO_UNICODE[36534] := 16#E8AC;
   // GBK_TO_UNICODE[36535] := 16#748E;
   // GBK_TO_UNICODE[36536] := 16#E8AD;
   // GBK_TO_UNICODE[36537] := 16#7480;
   // GBK_TO_UNICODE[36538] := 16#E8AE;
   // GBK_TO_UNICODE[36539] := 16#7481;
   // GBK_TO_UNICODE[36540] := 16#E8AF;
   // GBK_TO_UNICODE[36541] := 16#7487;
   // GBK_TO_UNICODE[36542] := 16#E8B0;
   // GBK_TO_UNICODE[36543] := 16#748B;
   // GBK_TO_UNICODE[36544] := 16#E8B1;
   // GBK_TO_UNICODE[36545] := 16#749E;
   // GBK_TO_UNICODE[36546] := 16#E8B2;
   // GBK_TO_UNICODE[36547] := 16#74A8;
   // GBK_TO_UNICODE[36548] := 16#E8B3;
   // GBK_TO_UNICODE[36549] := 16#74A9;
   // GBK_TO_UNICODE[36550] := 16#E8B4;
   // GBK_TO_UNICODE[36551] := 16#7490;
   // GBK_TO_UNICODE[36552] := 16#E8B5;
   // GBK_TO_UNICODE[36553] := 16#74A7;
   // GBK_TO_UNICODE[36554] := 16#E8B6;
   // GBK_TO_UNICODE[36555] := 16#74D2;
   // GBK_TO_UNICODE[36556] := 16#E8B7;
   // GBK_TO_UNICODE[36557] := 16#74BA;
   // GBK_TO_UNICODE[36558] := 16#E8B8;
   // GBK_TO_UNICODE[36559] := 16#97EA;
   // GBK_TO_UNICODE[36560] := 16#E8B9;
   // GBK_TO_UNICODE[36561] := 16#97EB;
   // GBK_TO_UNICODE[36562] := 16#E8BA;
   // GBK_TO_UNICODE[36563] := 16#97EC;
   // GBK_TO_UNICODE[36564] := 16#E8BB;
   // GBK_TO_UNICODE[36565] := 16#674C;
   // GBK_TO_UNICODE[36566] := 16#E8BC;
   // GBK_TO_UNICODE[36567] := 16#6753;
   // GBK_TO_UNICODE[36568] := 16#E8BD;
   // GBK_TO_UNICODE[36569] := 16#675E;
   // GBK_TO_UNICODE[36570] := 16#E8BE;
   // GBK_TO_UNICODE[36571] := 16#6748;
   // GBK_TO_UNICODE[36572] := 16#E8BF;
   // GBK_TO_UNICODE[36573] := 16#6769;
   // GBK_TO_UNICODE[36574] := 16#E8C0;
   // GBK_TO_UNICODE[36575] := 16#67A5;
   // GBK_TO_UNICODE[36576] := 16#E8C1;
   // GBK_TO_UNICODE[36577] := 16#6787;
   // GBK_TO_UNICODE[36578] := 16#E8C2;
   // GBK_TO_UNICODE[36579] := 16#676A;
   // GBK_TO_UNICODE[36580] := 16#E8C3;
   // GBK_TO_UNICODE[36581] := 16#6773;
   // GBK_TO_UNICODE[36582] := 16#E8C4;
   // GBK_TO_UNICODE[36583] := 16#6798;
   // GBK_TO_UNICODE[36584] := 16#E8C5;
   // GBK_TO_UNICODE[36585] := 16#67A7;
   // GBK_TO_UNICODE[36586] := 16#E8C6;
   // GBK_TO_UNICODE[36587] := 16#6775;
   // GBK_TO_UNICODE[36588] := 16#E8C7;
   // GBK_TO_UNICODE[36589] := 16#67A8;
   // GBK_TO_UNICODE[36590] := 16#E8C8;
   // GBK_TO_UNICODE[36591] := 16#679E;
   // GBK_TO_UNICODE[36592] := 16#E8C9;
   // GBK_TO_UNICODE[36593] := 16#67AD;
   // GBK_TO_UNICODE[36594] := 16#E8CA;
   // GBK_TO_UNICODE[36595] := 16#678B;
   // GBK_TO_UNICODE[36596] := 16#E8CB;
   // GBK_TO_UNICODE[36597] := 16#6777;
   // GBK_TO_UNICODE[36598] := 16#E8CC;
   // GBK_TO_UNICODE[36599] := 16#677C;
   // GBK_TO_UNICODE[36600] := 16#E8CD;
   // GBK_TO_UNICODE[36601] := 16#67F0;
   // GBK_TO_UNICODE[36602] := 16#E8CE;
   // GBK_TO_UNICODE[36603] := 16#6809;
   // GBK_TO_UNICODE[36604] := 16#E8CF;
   // GBK_TO_UNICODE[36605] := 16#67D8;
   // GBK_TO_UNICODE[36606] := 16#E8D0;
   // GBK_TO_UNICODE[36607] := 16#680A;
   // GBK_TO_UNICODE[36608] := 16#E8D1;
   // GBK_TO_UNICODE[36609] := 16#67E9;
   // GBK_TO_UNICODE[36610] := 16#E8D2;
   // GBK_TO_UNICODE[36611] := 16#67B0;
   // GBK_TO_UNICODE[36612] := 16#E8D3;
   // GBK_TO_UNICODE[36613] := 16#680C;
   // GBK_TO_UNICODE[36614] := 16#E8D4;
   // GBK_TO_UNICODE[36615] := 16#67D9;
   // GBK_TO_UNICODE[36616] := 16#E8D5;
   // GBK_TO_UNICODE[36617] := 16#67B5;
   // GBK_TO_UNICODE[36618] := 16#E8D6;
   // GBK_TO_UNICODE[36619] := 16#67DA;
   // GBK_TO_UNICODE[36620] := 16#E8D7;
   // GBK_TO_UNICODE[36621] := 16#67B3;
   // GBK_TO_UNICODE[36622] := 16#E8D8;
   // GBK_TO_UNICODE[36623] := 16#67DD;
   // GBK_TO_UNICODE[36624] := 16#E8D9;
   // GBK_TO_UNICODE[36625] := 16#6800;
   // GBK_TO_UNICODE[36626] := 16#E8DA;
   // GBK_TO_UNICODE[36627] := 16#67C3;
   // GBK_TO_UNICODE[36628] := 16#E8DB;
   // GBK_TO_UNICODE[36629] := 16#67B8;
   // GBK_TO_UNICODE[36630] := 16#E8DC;
   // GBK_TO_UNICODE[36631] := 16#67E2;
   // GBK_TO_UNICODE[36632] := 16#E8DD;
   // GBK_TO_UNICODE[36633] := 16#680E;
   // GBK_TO_UNICODE[36634] := 16#E8DE;
   // GBK_TO_UNICODE[36635] := 16#67C1;
   // GBK_TO_UNICODE[36636] := 16#E8DF;
   // GBK_TO_UNICODE[36637] := 16#67FD;
   // GBK_TO_UNICODE[36638] := 16#E8E0;
   // GBK_TO_UNICODE[36639] := 16#6832;
   // GBK_TO_UNICODE[36640] := 16#E8E1;
   // GBK_TO_UNICODE[36641] := 16#6833;
   // GBK_TO_UNICODE[36642] := 16#E8E2;
   // GBK_TO_UNICODE[36643] := 16#6860;
   // GBK_TO_UNICODE[36644] := 16#E8E3;
   // GBK_TO_UNICODE[36645] := 16#6861;
   // GBK_TO_UNICODE[36646] := 16#E8E4;
   // GBK_TO_UNICODE[36647] := 16#684E;
   // GBK_TO_UNICODE[36648] := 16#E8E5;
   // GBK_TO_UNICODE[36649] := 16#6862;
   // GBK_TO_UNICODE[36650] := 16#E8E6;
   // GBK_TO_UNICODE[36651] := 16#6844;
   // GBK_TO_UNICODE[36652] := 16#E8E7;
   // GBK_TO_UNICODE[36653] := 16#6864;
   // GBK_TO_UNICODE[36654] := 16#E8E8;
   // GBK_TO_UNICODE[36655] := 16#6883;
   // GBK_TO_UNICODE[36656] := 16#E8E9;
   // GBK_TO_UNICODE[36657] := 16#681D;
   // GBK_TO_UNICODE[36658] := 16#E8EA;
   // GBK_TO_UNICODE[36659] := 16#6855;
   // GBK_TO_UNICODE[36660] := 16#E8EB;
   // GBK_TO_UNICODE[36661] := 16#6866;
   // GBK_TO_UNICODE[36662] := 16#E8EC;
   // GBK_TO_UNICODE[36663] := 16#6841;
   // GBK_TO_UNICODE[36664] := 16#E8ED;
   // GBK_TO_UNICODE[36665] := 16#6867;
   // GBK_TO_UNICODE[36666] := 16#E8EE;
   // GBK_TO_UNICODE[36667] := 16#6840;
   // GBK_TO_UNICODE[36668] := 16#E8EF;
   // GBK_TO_UNICODE[36669] := 16#683E;
   // GBK_TO_UNICODE[36670] := 16#E8F0;
   // GBK_TO_UNICODE[36671] := 16#684A;
   // GBK_TO_UNICODE[36672] := 16#E8F1;
   // GBK_TO_UNICODE[36673] := 16#6849;
   // GBK_TO_UNICODE[36674] := 16#E8F2;
   // GBK_TO_UNICODE[36675] := 16#6829;
   // GBK_TO_UNICODE[36676] := 16#E8F3;
   // GBK_TO_UNICODE[36677] := 16#68B5;
   // GBK_TO_UNICODE[36678] := 16#E8F4;
   // GBK_TO_UNICODE[36679] := 16#688F;
   // GBK_TO_UNICODE[36680] := 16#E8F5;
   // GBK_TO_UNICODE[36681] := 16#6874;
   // GBK_TO_UNICODE[36682] := 16#E8F6;
   // GBK_TO_UNICODE[36683] := 16#6877;
   // GBK_TO_UNICODE[36684] := 16#E8F7;
   // GBK_TO_UNICODE[36685] := 16#6893;
   // GBK_TO_UNICODE[36686] := 16#E8F8;
   // GBK_TO_UNICODE[36687] := 16#686B;
   // GBK_TO_UNICODE[36688] := 16#E8F9;
   // GBK_TO_UNICODE[36689] := 16#68C2;
   // GBK_TO_UNICODE[36690] := 16#E8FA;
   // GBK_TO_UNICODE[36691] := 16#696E;
   // GBK_TO_UNICODE[36692] := 16#E8FB;
   // GBK_TO_UNICODE[36693] := 16#68FC;
   // GBK_TO_UNICODE[36694] := 16#E8FC;
   // GBK_TO_UNICODE[36695] := 16#691F;
   // GBK_TO_UNICODE[36696] := 16#E8FD;
   // GBK_TO_UNICODE[36697] := 16#6920;
   // GBK_TO_UNICODE[36698] := 16#E8FE;
   // GBK_TO_UNICODE[36699] := 16#68F9;
   // GBK_TO_UNICODE[36700] := 16#E940;
   // GBK_TO_UNICODE[36701] := 16#9527;
   // GBK_TO_UNICODE[36702] := 16#E941;
   // GBK_TO_UNICODE[36703] := 16#9533;
   // GBK_TO_UNICODE[36704] := 16#E942;
   // GBK_TO_UNICODE[36705] := 16#953D;
   // GBK_TO_UNICODE[36706] := 16#E943;
   // GBK_TO_UNICODE[36707] := 16#9543;
   // GBK_TO_UNICODE[36708] := 16#E944;
   // GBK_TO_UNICODE[36709] := 16#9548;
   // GBK_TO_UNICODE[36710] := 16#E945;
   // GBK_TO_UNICODE[36711] := 16#954B;
   // GBK_TO_UNICODE[36712] := 16#E946;
   // GBK_TO_UNICODE[36713] := 16#9555;
   // GBK_TO_UNICODE[36714] := 16#E947;
   // GBK_TO_UNICODE[36715] := 16#955A;
   // GBK_TO_UNICODE[36716] := 16#E948;
   // GBK_TO_UNICODE[36717] := 16#9560;
   // GBK_TO_UNICODE[36718] := 16#E949;
   // GBK_TO_UNICODE[36719] := 16#956E;
   // GBK_TO_UNICODE[36720] := 16#E94A;
   // GBK_TO_UNICODE[36721] := 16#9574;
   // GBK_TO_UNICODE[36722] := 16#E94B;
   // GBK_TO_UNICODE[36723] := 16#9575;
   // GBK_TO_UNICODE[36724] := 16#E94C;
   // GBK_TO_UNICODE[36725] := 16#9577;
   // GBK_TO_UNICODE[36726] := 16#E94D;
   // GBK_TO_UNICODE[36727] := 16#9578;
   // GBK_TO_UNICODE[36728] := 16#E94E;
   // GBK_TO_UNICODE[36729] := 16#9579;
   // GBK_TO_UNICODE[36730] := 16#E94F;
   // GBK_TO_UNICODE[36731] := 16#957A;
   // GBK_TO_UNICODE[36732] := 16#E950;
   // GBK_TO_UNICODE[36733] := 16#957B;
   // GBK_TO_UNICODE[36734] := 16#E951;
   // GBK_TO_UNICODE[36735] := 16#957C;
   // GBK_TO_UNICODE[36736] := 16#E952;
   // GBK_TO_UNICODE[36737] := 16#957D;
   // GBK_TO_UNICODE[36738] := 16#E953;
   // GBK_TO_UNICODE[36739] := 16#957E;
   // GBK_TO_UNICODE[36740] := 16#E954;
   // GBK_TO_UNICODE[36741] := 16#9580;
   // GBK_TO_UNICODE[36742] := 16#E955;
   // GBK_TO_UNICODE[36743] := 16#9581;
   // GBK_TO_UNICODE[36744] := 16#E956;
   // GBK_TO_UNICODE[36745] := 16#9582;
   // GBK_TO_UNICODE[36746] := 16#E957;
   // GBK_TO_UNICODE[36747] := 16#9583;
   // GBK_TO_UNICODE[36748] := 16#E958;
   // GBK_TO_UNICODE[36749] := 16#9584;
   // GBK_TO_UNICODE[36750] := 16#E959;
   // GBK_TO_UNICODE[36751] := 16#9585;
   // GBK_TO_UNICODE[36752] := 16#E95A;
   // GBK_TO_UNICODE[36753] := 16#9586;
   // GBK_TO_UNICODE[36754] := 16#E95B;
   // GBK_TO_UNICODE[36755] := 16#9587;
   // GBK_TO_UNICODE[36756] := 16#E95C;
   // GBK_TO_UNICODE[36757] := 16#9588;
   // GBK_TO_UNICODE[36758] := 16#E95D;
   // GBK_TO_UNICODE[36759] := 16#9589;
   // GBK_TO_UNICODE[36760] := 16#E95E;
   // GBK_TO_UNICODE[36761] := 16#958A;
   // GBK_TO_UNICODE[36762] := 16#E95F;
   // GBK_TO_UNICODE[36763] := 16#958B;
   // GBK_TO_UNICODE[36764] := 16#E960;
   // GBK_TO_UNICODE[36765] := 16#958C;
   // GBK_TO_UNICODE[36766] := 16#E961;
   // GBK_TO_UNICODE[36767] := 16#958D;
   // GBK_TO_UNICODE[36768] := 16#E962;
   // GBK_TO_UNICODE[36769] := 16#958E;
   // GBK_TO_UNICODE[36770] := 16#E963;
   // GBK_TO_UNICODE[36771] := 16#958F;
   // GBK_TO_UNICODE[36772] := 16#E964;
   // GBK_TO_UNICODE[36773] := 16#9590;
   // GBK_TO_UNICODE[36774] := 16#E965;
   // GBK_TO_UNICODE[36775] := 16#9591;
   // GBK_TO_UNICODE[36776] := 16#E966;
   // GBK_TO_UNICODE[36777] := 16#9592;
   // GBK_TO_UNICODE[36778] := 16#E967;
   // GBK_TO_UNICODE[36779] := 16#9593;
   // GBK_TO_UNICODE[36780] := 16#E968;
   // GBK_TO_UNICODE[36781] := 16#9594;
   // GBK_TO_UNICODE[36782] := 16#E969;
   // GBK_TO_UNICODE[36783] := 16#9595;
   // GBK_TO_UNICODE[36784] := 16#E96A;
   // GBK_TO_UNICODE[36785] := 16#9596;
   // GBK_TO_UNICODE[36786] := 16#E96B;
   // GBK_TO_UNICODE[36787] := 16#9597;
   // GBK_TO_UNICODE[36788] := 16#E96C;
   // GBK_TO_UNICODE[36789] := 16#9598;
   // GBK_TO_UNICODE[36790] := 16#E96D;
   // GBK_TO_UNICODE[36791] := 16#9599;
   // GBK_TO_UNICODE[36792] := 16#E96E;
   // GBK_TO_UNICODE[36793] := 16#959A;
   // GBK_TO_UNICODE[36794] := 16#E96F;
   // GBK_TO_UNICODE[36795] := 16#959B;
   // GBK_TO_UNICODE[36796] := 16#E970;
   // GBK_TO_UNICODE[36797] := 16#959C;
   // GBK_TO_UNICODE[36798] := 16#E971;
   // GBK_TO_UNICODE[36799] := 16#959D;
   // GBK_TO_UNICODE[36800] := 16#E972;
   // GBK_TO_UNICODE[36801] := 16#959E;
   // GBK_TO_UNICODE[36802] := 16#E973;
   // GBK_TO_UNICODE[36803] := 16#959F;
   // GBK_TO_UNICODE[36804] := 16#E974;
   // GBK_TO_UNICODE[36805] := 16#95A0;
   // GBK_TO_UNICODE[36806] := 16#E975;
   // GBK_TO_UNICODE[36807] := 16#95A1;
   // GBK_TO_UNICODE[36808] := 16#E976;
   // GBK_TO_UNICODE[36809] := 16#95A2;
   // GBK_TO_UNICODE[36810] := 16#E977;
   // GBK_TO_UNICODE[36811] := 16#95A3;
   // GBK_TO_UNICODE[36812] := 16#E978;
   // GBK_TO_UNICODE[36813] := 16#95A4;
   // GBK_TO_UNICODE[36814] := 16#E979;
   // GBK_TO_UNICODE[36815] := 16#95A5;
   // GBK_TO_UNICODE[36816] := 16#E97A;
   // GBK_TO_UNICODE[36817] := 16#95A6;
   // GBK_TO_UNICODE[36818] := 16#E97B;
   // GBK_TO_UNICODE[36819] := 16#95A7;
   // GBK_TO_UNICODE[36820] := 16#E97C;
   // GBK_TO_UNICODE[36821] := 16#95A8;
   // GBK_TO_UNICODE[36822] := 16#E97D;
   // GBK_TO_UNICODE[36823] := 16#95A9;
   // GBK_TO_UNICODE[36824] := 16#E97E;
   // GBK_TO_UNICODE[36825] := 16#95AA;
   // GBK_TO_UNICODE[36826] := 16#E980;
   // GBK_TO_UNICODE[36827] := 16#95AB;
   // GBK_TO_UNICODE[36828] := 16#E981;
   // GBK_TO_UNICODE[36829] := 16#95AC;
   // GBK_TO_UNICODE[36830] := 16#E982;
   // GBK_TO_UNICODE[36831] := 16#95AD;
   // GBK_TO_UNICODE[36832] := 16#E983;
   // GBK_TO_UNICODE[36833] := 16#95AE;
   // GBK_TO_UNICODE[36834] := 16#E984;
   // GBK_TO_UNICODE[36835] := 16#95AF;
   // GBK_TO_UNICODE[36836] := 16#E985;
   // GBK_TO_UNICODE[36837] := 16#95B0;
   // GBK_TO_UNICODE[36838] := 16#E986;
   // GBK_TO_UNICODE[36839] := 16#95B1;
   // GBK_TO_UNICODE[36840] := 16#E987;
   // GBK_TO_UNICODE[36841] := 16#95B2;
   // GBK_TO_UNICODE[36842] := 16#E988;
   // GBK_TO_UNICODE[36843] := 16#95B3;
   // GBK_TO_UNICODE[36844] := 16#E989;
   // GBK_TO_UNICODE[36845] := 16#95B4;
   // GBK_TO_UNICODE[36846] := 16#E98A;
   // GBK_TO_UNICODE[36847] := 16#95B5;
   // GBK_TO_UNICODE[36848] := 16#E98B;
   // GBK_TO_UNICODE[36849] := 16#95B6;
   // GBK_TO_UNICODE[36850] := 16#E98C;
   // GBK_TO_UNICODE[36851] := 16#95B7;
   // GBK_TO_UNICODE[36852] := 16#E98D;
   // GBK_TO_UNICODE[36853] := 16#95B8;
   // GBK_TO_UNICODE[36854] := 16#E98E;
   // GBK_TO_UNICODE[36855] := 16#95B9;
   // GBK_TO_UNICODE[36856] := 16#E98F;
   // GBK_TO_UNICODE[36857] := 16#95BA;
   // GBK_TO_UNICODE[36858] := 16#E990;
   // GBK_TO_UNICODE[36859] := 16#95BB;
   // GBK_TO_UNICODE[36860] := 16#E991;
   // GBK_TO_UNICODE[36861] := 16#95BC;
   // GBK_TO_UNICODE[36862] := 16#E992;
   // GBK_TO_UNICODE[36863] := 16#95BD;
   // GBK_TO_UNICODE[36864] := 16#E993;
   // GBK_TO_UNICODE[36865] := 16#95BE;
   // GBK_TO_UNICODE[36866] := 16#E994;
   // GBK_TO_UNICODE[36867] := 16#95BF;
   // GBK_TO_UNICODE[36868] := 16#E995;
   // GBK_TO_UNICODE[36869] := 16#95C0;
   // GBK_TO_UNICODE[36870] := 16#E996;
   // GBK_TO_UNICODE[36871] := 16#95C1;
   // GBK_TO_UNICODE[36872] := 16#E997;
   // GBK_TO_UNICODE[36873] := 16#95C2;
   // GBK_TO_UNICODE[36874] := 16#E998;
   // GBK_TO_UNICODE[36875] := 16#95C3;
   // GBK_TO_UNICODE[36876] := 16#E999;
   // GBK_TO_UNICODE[36877] := 16#95C4;
   // GBK_TO_UNICODE[36878] := 16#E99A;
   // GBK_TO_UNICODE[36879] := 16#95C5;
   // GBK_TO_UNICODE[36880] := 16#E99B;
   // GBK_TO_UNICODE[36881] := 16#95C6;
   // GBK_TO_UNICODE[36882] := 16#E99C;
   // GBK_TO_UNICODE[36883] := 16#95C7;
   // GBK_TO_UNICODE[36884] := 16#E99D;
   // GBK_TO_UNICODE[36885] := 16#95C8;
   // GBK_TO_UNICODE[36886] := 16#E99E;
   // GBK_TO_UNICODE[36887] := 16#95C9;
   // GBK_TO_UNICODE[36888] := 16#E99F;
   // GBK_TO_UNICODE[36889] := 16#95CA;
   // GBK_TO_UNICODE[36890] := 16#E9A0;
   // GBK_TO_UNICODE[36891] := 16#95CB;
   // GBK_TO_UNICODE[36892] := 16#E9A1;
   // GBK_TO_UNICODE[36893] := 16#6924;
   // GBK_TO_UNICODE[36894] := 16#E9A2;
   // GBK_TO_UNICODE[36895] := 16#68F0;
   // GBK_TO_UNICODE[36896] := 16#E9A3;
   // GBK_TO_UNICODE[36897] := 16#690B;
   // GBK_TO_UNICODE[36898] := 16#E9A4;
   // GBK_TO_UNICODE[36899] := 16#6901;
   // GBK_TO_UNICODE[36900] := 16#E9A5;
   // GBK_TO_UNICODE[36901] := 16#6957;
   // GBK_TO_UNICODE[36902] := 16#E9A6;
   // GBK_TO_UNICODE[36903] := 16#68E3;
   // GBK_TO_UNICODE[36904] := 16#E9A7;
   // GBK_TO_UNICODE[36905] := 16#6910;
   // GBK_TO_UNICODE[36906] := 16#E9A8;
   // GBK_TO_UNICODE[36907] := 16#6971;
   // GBK_TO_UNICODE[36908] := 16#E9A9;
   // GBK_TO_UNICODE[36909] := 16#6939;
   // GBK_TO_UNICODE[36910] := 16#E9AA;
   // GBK_TO_UNICODE[36911] := 16#6960;
   // GBK_TO_UNICODE[36912] := 16#E9AB;
   // GBK_TO_UNICODE[36913] := 16#6942;
   // GBK_TO_UNICODE[36914] := 16#E9AC;
   // GBK_TO_UNICODE[36915] := 16#695D;
   // GBK_TO_UNICODE[36916] := 16#E9AD;
   // GBK_TO_UNICODE[36917] := 16#6984;
   // GBK_TO_UNICODE[36918] := 16#E9AE;
   // GBK_TO_UNICODE[36919] := 16#696B;
   // GBK_TO_UNICODE[36920] := 16#E9AF;
   // GBK_TO_UNICODE[36921] := 16#6980;
   // GBK_TO_UNICODE[36922] := 16#E9B0;
   // GBK_TO_UNICODE[36923] := 16#6998;
   // GBK_TO_UNICODE[36924] := 16#E9B1;
   // GBK_TO_UNICODE[36925] := 16#6978;
   // GBK_TO_UNICODE[36926] := 16#E9B2;
   // GBK_TO_UNICODE[36927] := 16#6934;
   // GBK_TO_UNICODE[36928] := 16#E9B3;
   // GBK_TO_UNICODE[36929] := 16#69CC;
   // GBK_TO_UNICODE[36930] := 16#E9B4;
   // GBK_TO_UNICODE[36931] := 16#6987;
   // GBK_TO_UNICODE[36932] := 16#E9B5;
   // GBK_TO_UNICODE[36933] := 16#6988;
   // GBK_TO_UNICODE[36934] := 16#E9B6;
   // GBK_TO_UNICODE[36935] := 16#69CE;
   // GBK_TO_UNICODE[36936] := 16#E9B7;
   // GBK_TO_UNICODE[36937] := 16#6989;
   // GBK_TO_UNICODE[36938] := 16#E9B8;
   // GBK_TO_UNICODE[36939] := 16#6966;
   // GBK_TO_UNICODE[36940] := 16#E9B9;
   // GBK_TO_UNICODE[36941] := 16#6963;
   // GBK_TO_UNICODE[36942] := 16#E9BA;
   // GBK_TO_UNICODE[36943] := 16#6979;
   // GBK_TO_UNICODE[36944] := 16#E9BB;
   // GBK_TO_UNICODE[36945] := 16#699B;
   // GBK_TO_UNICODE[36946] := 16#E9BC;
   // GBK_TO_UNICODE[36947] := 16#69A7;
   // GBK_TO_UNICODE[36948] := 16#E9BD;
   // GBK_TO_UNICODE[36949] := 16#69BB;
   // GBK_TO_UNICODE[36950] := 16#E9BE;
   // GBK_TO_UNICODE[36951] := 16#69AB;
   // GBK_TO_UNICODE[36952] := 16#E9BF;
   // GBK_TO_UNICODE[36953] := 16#69AD;
   // GBK_TO_UNICODE[36954] := 16#E9C0;
   // GBK_TO_UNICODE[36955] := 16#69D4;
   // GBK_TO_UNICODE[36956] := 16#E9C1;
   // GBK_TO_UNICODE[36957] := 16#69B1;
   // GBK_TO_UNICODE[36958] := 16#E9C2;
   // GBK_TO_UNICODE[36959] := 16#69C1;
   // GBK_TO_UNICODE[36960] := 16#E9C3;
   // GBK_TO_UNICODE[36961] := 16#69CA;
   // GBK_TO_UNICODE[36962] := 16#E9C4;
   // GBK_TO_UNICODE[36963] := 16#69DF;
   // GBK_TO_UNICODE[36964] := 16#E9C5;
   // GBK_TO_UNICODE[36965] := 16#6995;
   // GBK_TO_UNICODE[36966] := 16#E9C6;
   // GBK_TO_UNICODE[36967] := 16#69E0;
   // GBK_TO_UNICODE[36968] := 16#E9C7;
   // GBK_TO_UNICODE[36969] := 16#698D;
   // GBK_TO_UNICODE[36970] := 16#E9C8;
   // GBK_TO_UNICODE[36971] := 16#69FF;
   // GBK_TO_UNICODE[36972] := 16#E9C9;
   // GBK_TO_UNICODE[36973] := 16#6A2F;
   // GBK_TO_UNICODE[36974] := 16#E9CA;
   // GBK_TO_UNICODE[36975] := 16#69ED;
   // GBK_TO_UNICODE[36976] := 16#E9CB;
   // GBK_TO_UNICODE[36977] := 16#6A17;
   // GBK_TO_UNICODE[36978] := 16#E9CC;
   // GBK_TO_UNICODE[36979] := 16#6A18;
   // GBK_TO_UNICODE[36980] := 16#E9CD;
   // GBK_TO_UNICODE[36981] := 16#6A65;
   // GBK_TO_UNICODE[36982] := 16#E9CE;
   // GBK_TO_UNICODE[36983] := 16#69F2;
   // GBK_TO_UNICODE[36984] := 16#E9CF;
   // GBK_TO_UNICODE[36985] := 16#6A44;
   // GBK_TO_UNICODE[36986] := 16#E9D0;
   // GBK_TO_UNICODE[36987] := 16#6A3E;
   // GBK_TO_UNICODE[36988] := 16#E9D1;
   // GBK_TO_UNICODE[36989] := 16#6AA0;
   // GBK_TO_UNICODE[36990] := 16#E9D2;
   // GBK_TO_UNICODE[36991] := 16#6A50;
   // GBK_TO_UNICODE[36992] := 16#E9D3;
   // GBK_TO_UNICODE[36993] := 16#6A5B;
   // GBK_TO_UNICODE[36994] := 16#E9D4;
   // GBK_TO_UNICODE[36995] := 16#6A35;
   // GBK_TO_UNICODE[36996] := 16#E9D5;
   // GBK_TO_UNICODE[36997] := 16#6A8E;
   // GBK_TO_UNICODE[36998] := 16#E9D6;
   // GBK_TO_UNICODE[36999] := 16#6A79;
   // GBK_TO_UNICODE[37000] := 16#E9D7;
   // GBK_TO_UNICODE[37001] := 16#6A3D;
   // GBK_TO_UNICODE[37002] := 16#E9D8;
   // GBK_TO_UNICODE[37003] := 16#6A28;
   // GBK_TO_UNICODE[37004] := 16#E9D9;
   // GBK_TO_UNICODE[37005] := 16#6A58;
   // GBK_TO_UNICODE[37006] := 16#E9DA;
   // GBK_TO_UNICODE[37007] := 16#6A7C;
   // GBK_TO_UNICODE[37008] := 16#E9DB;
   // GBK_TO_UNICODE[37009] := 16#6A91;
   // GBK_TO_UNICODE[37010] := 16#E9DC;
   // GBK_TO_UNICODE[37011] := 16#6A90;
   // GBK_TO_UNICODE[37012] := 16#E9DD;
   // GBK_TO_UNICODE[37013] := 16#6AA9;
   // GBK_TO_UNICODE[37014] := 16#E9DE;
   // GBK_TO_UNICODE[37015] := 16#6A97;
   // GBK_TO_UNICODE[37016] := 16#E9DF;
   // GBK_TO_UNICODE[37017] := 16#6AAB;
   // GBK_TO_UNICODE[37018] := 16#E9E0;
   // GBK_TO_UNICODE[37019] := 16#7337;
   // GBK_TO_UNICODE[37020] := 16#E9E1;
   // GBK_TO_UNICODE[37021] := 16#7352;
   // GBK_TO_UNICODE[37022] := 16#E9E2;
   // GBK_TO_UNICODE[37023] := 16#6B81;
   // GBK_TO_UNICODE[37024] := 16#E9E3;
   // GBK_TO_UNICODE[37025] := 16#6B82;
   // GBK_TO_UNICODE[37026] := 16#E9E4;
   // GBK_TO_UNICODE[37027] := 16#6B87;
   // GBK_TO_UNICODE[37028] := 16#E9E5;
   // GBK_TO_UNICODE[37029] := 16#6B84;
   // GBK_TO_UNICODE[37030] := 16#E9E6;
   // GBK_TO_UNICODE[37031] := 16#6B92;
   // GBK_TO_UNICODE[37032] := 16#E9E7;
   // GBK_TO_UNICODE[37033] := 16#6B93;
   // GBK_TO_UNICODE[37034] := 16#E9E8;
   // GBK_TO_UNICODE[37035] := 16#6B8D;
   // GBK_TO_UNICODE[37036] := 16#E9E9;
   // GBK_TO_UNICODE[37037] := 16#6B9A;
   // GBK_TO_UNICODE[37038] := 16#E9EA;
   // GBK_TO_UNICODE[37039] := 16#6B9B;
   // GBK_TO_UNICODE[37040] := 16#E9EB;
   // GBK_TO_UNICODE[37041] := 16#6BA1;
   // GBK_TO_UNICODE[37042] := 16#E9EC;
   // GBK_TO_UNICODE[37043] := 16#6BAA;
   // GBK_TO_UNICODE[37044] := 16#E9ED;
   // GBK_TO_UNICODE[37045] := 16#8F6B;
   // GBK_TO_UNICODE[37046] := 16#E9EE;
   // GBK_TO_UNICODE[37047] := 16#8F6D;
   // GBK_TO_UNICODE[37048] := 16#E9EF;
   // GBK_TO_UNICODE[37049] := 16#8F71;
   // GBK_TO_UNICODE[37050] := 16#E9F0;
   // GBK_TO_UNICODE[37051] := 16#8F72;
   // GBK_TO_UNICODE[37052] := 16#E9F1;
   // GBK_TO_UNICODE[37053] := 16#8F73;
   // GBK_TO_UNICODE[37054] := 16#E9F2;
   // GBK_TO_UNICODE[37055] := 16#8F75;
   // GBK_TO_UNICODE[37056] := 16#E9F3;
   // GBK_TO_UNICODE[37057] := 16#8F76;
   // GBK_TO_UNICODE[37058] := 16#E9F4;
   // GBK_TO_UNICODE[37059] := 16#8F78;
   // GBK_TO_UNICODE[37060] := 16#E9F5;
   // GBK_TO_UNICODE[37061] := 16#8F77;
   // GBK_TO_UNICODE[37062] := 16#E9F6;
   // GBK_TO_UNICODE[37063] := 16#8F79;
   // GBK_TO_UNICODE[37064] := 16#E9F7;
   // GBK_TO_UNICODE[37065] := 16#8F7A;
   // GBK_TO_UNICODE[37066] := 16#E9F8;
   // GBK_TO_UNICODE[37067] := 16#8F7C;
